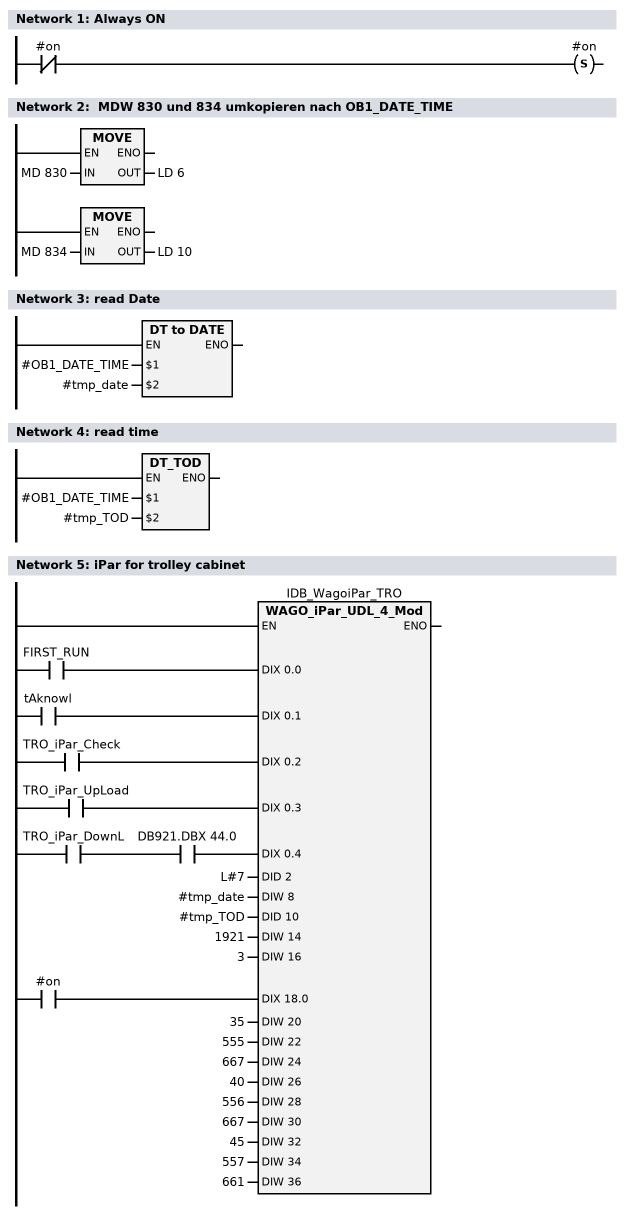
[picture p333: iPar_ServerCall networks 1-5]
NETWORK
TITLE = Always ON
      AN    #on;
      S     #on;
NETWORK
TITLE =  MDW 830 und 834 umkopieren nach OB1_DATE_TIME
      L     MD 830;
      T     LD 6;
      L     MD 834;
      T     LD 10;
NETWORK
TITLE = read Date
      CALL  "DT to DATE" (
           $1                       := #OB1_DATE_TIME,
           $2                       := #tmp_date);
      NOP   0;
NETWORK
TITLE = read time
      CALL  "DT_TOD" (
           $1                       := #OB1_DATE_TIME,
           $2                       := #tmp_TOD);
      NOP   0;
NETWORK
TITLE = iPar for trolley cabinet
      A     "FIRST_RUN";
      =     L 15.0;
      BLD   103;
      A     "tAknowl";
      =     L 15.1;
      BLD   103;
      A     "TRO_iPar_Check";
      =     L 15.2;
      BLD   103;
      A     "TRO_iPar_UpLoad";
      =     L 15.3;
      BLD   103;
      A     "TRO_iPar_DownL";
      A     DB921.DBX 44.0;
      =     L 15.4;
      BLD   103;
      A     #on;
      =     L 16.0;
      BLD   103;
      CALL  "WAGO_iPar_UDL_4_Mod" , "IDB_WagoiPar_TRO" (
           DIX 0.0                  := L 15.0,
           DIX 0.1                  := L 15.1,
           DIX 0.2                  := L 15.2,
           DIX 0.3                  := L 15.3,
           DIX 0.4                  := L 15.4,
           DID 2                    := L#7,
           DIW 8                    := #tmp_date,
           DID 10                   := #tmp_TOD,
           DIW 14                   := 1921,
           DIW 16                   := 3,
           DIX 18.0                 := L 16.0,
           DIW 20                   := 35,
           DIW 22                   := 555,
           DIW 24                   := 667,
           DIW 26                   := 40,
           DIW 28                   := 556,
           DIW 30                   := 667,
           DIW 32                   := 45,
           DIW 34                   := 557,
           DIW 36                   := 661);
      NOP   0;
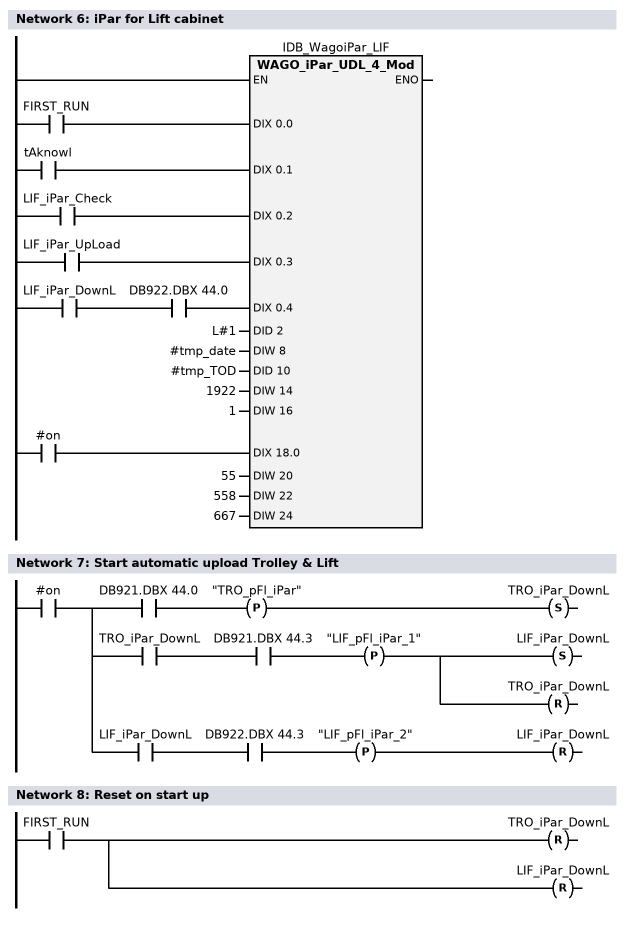
NETWORK
TITLE = iPar for Lift cabinet
      A     "FIRST_RUN";
      =     L 15.0;
      BLD   103;
      A     "tAknowl";
      =     L 15.1;
      BLD   103;
      A     "LIF_iPar_Check";
      =     L 15.2;
      BLD   103;
      A     "LIF_iPar_UpLoad";
      =     L 15.3;
      BLD   103;
      A     "LIF_iPar_DownL";
      A     DB922.DBX 44.0;
      =     L 15.4;
      BLD   103;
      A     #on;
      =     L 16.0;
      BLD   103;
      CALL  "WAGO_iPar_UDL_4_Mod" , "IDB_WagoiPar_LIF" (
           DIX 0.0                  := L 15.0,
           DIX 0.1                  := L 15.1,
           DIX 0.2                  := L 15.2,
           DIX 0.3                  := L 15.3,
           DIX 0.4                  := L 15.4,
           DID 2                    := L#1,
           DIW 8                    := #tmp_date,
           DID 10                   := #tmp_TOD,
           DIW 14                   := 1922,
           DIW 16                   := 1,
           DIX 18.0                 := L 16.0,
           DIW 20                   := 55,
           DIW 22                   := 558,
           DIW 24                   := 667);
      NOP   0;
NETWORK
TITLE = Start automatic upload Trolley & Lift
      A     #on;
      =     L 15.0;
      A     L 15.0;
      A     DB921.DBX 44.0;
      FP    "TRO_pFl_iPar";
      S     "TRO_iPar_DownL";
      A     L 15.0;
      A     "TRO_iPar_DownL";
      A     DB921.DBX 44.3;
      FP    "LIF_pFl_iPar_1";
      S     "LIF_iPar_DownL";
      R     "TRO_iPar_DownL";
      A     L 15.0;
      A     "LIF_iPar_DownL";
      A     DB922.DBX 44.3;
      FP    "LIF_pFl_iPar_2";
      R     "LIF_iPar_DownL";
NETWORK
TITLE = Reset on start up
      A     "FIRST_RUN";
      R     "TRO_iPar_DownL";
      R     "LIF_iPar_DownL";
END_FUNCTION

FUNCTION "Scan_LIF_New" : VOID	// FC 1025
TITLE = scan positions lift
VERSION : 1.0
VAR_INPUT
  in_x_ReleaseScan : BOOL ;
  in_i_LiDbNo_1 : INT ;
  in_i_LiDbNo_2 : INT ;
  in_di_NoOfDataSetsli : DINT ;
  in_di_DatSetLenghtli : DINT ;
  in_di_ActAxisPos : DINT ;
  in_di_AreaWin : DINT ;
  in_di_PosWin : DINT ;
  in_x_SelectDirection : BOOL ;	//1=right
END_VAR
VAR_OUTPUT
  out_di_Pointer : DINT ;
  out_i_DB_No : INT ;
  out_b_DB_dir_1 : BOOL ;
  out_b_DB_dir_2 : BOOL ;
  out_i_AreaNo : INT ;
  out_b_InArea : BOOL ;
  out_b_InPosHo : BOOL ;
  out_b_InPosHu : BOOL ;
  out_di_PosValHo : DINT ;
  out_di_PosValHu : DINT ;
  out_HookDataSet : UDT 102;
END_VAR
VAR_TEMP
  tmp_any_1 : ANY ;
  tmp_any_2 : ANY ;
  Save_AR1 : DWORD ;
  Save_AR2 : DWORD ;
  tmp_di_Pointer : DINT ;
  tmp_di_PosWinMinus : DINT ;
  tmp_di_PosWinPlus : DINT ;
  tmp_di_1 : DINT ;
  tmp_di_PosValHu_1 : DINT ;
  tmp_di_PosValHu_2 : DINT ;
  tmp_i_PosNo : INT ;
  tmp_i_Hooktype : INT ;
  tmp_i_DbNo : INT ;
  tmp_i_DbNo_2 : INT ;
  RetVal : INT ;
  ON : BOOL ;
  OFF : BOOL ;
  tmp_b_LoopBrake : BOOL ;
  tmp_b_1 : BOOL ;
  tmp_b_InArea_1 : BOOL ;
  tmp_b_InArea_2 : BOOL ;
  tmp_b_InPosHo_1 : BOOL ;
  tmp_b_InPosHo_2 : BOOL ;
  tmp_b_InPosHu_1 : BOOL ;
  tmp_b_InPosHu_2 : BOOL ;
  tmpHookDataSet_1 : UDT 102;
  tmpHookDataSet_2 : UDT 102;
END_VAR
BEGIN
NETWORK
TITLE = save register
      TAR1  #Save_AR1;
      TAR2  #Save_AR2;
NETWORK
TITLE = on/off
      SET;
      =     #ON;
      CLR;
      =     #OFF;
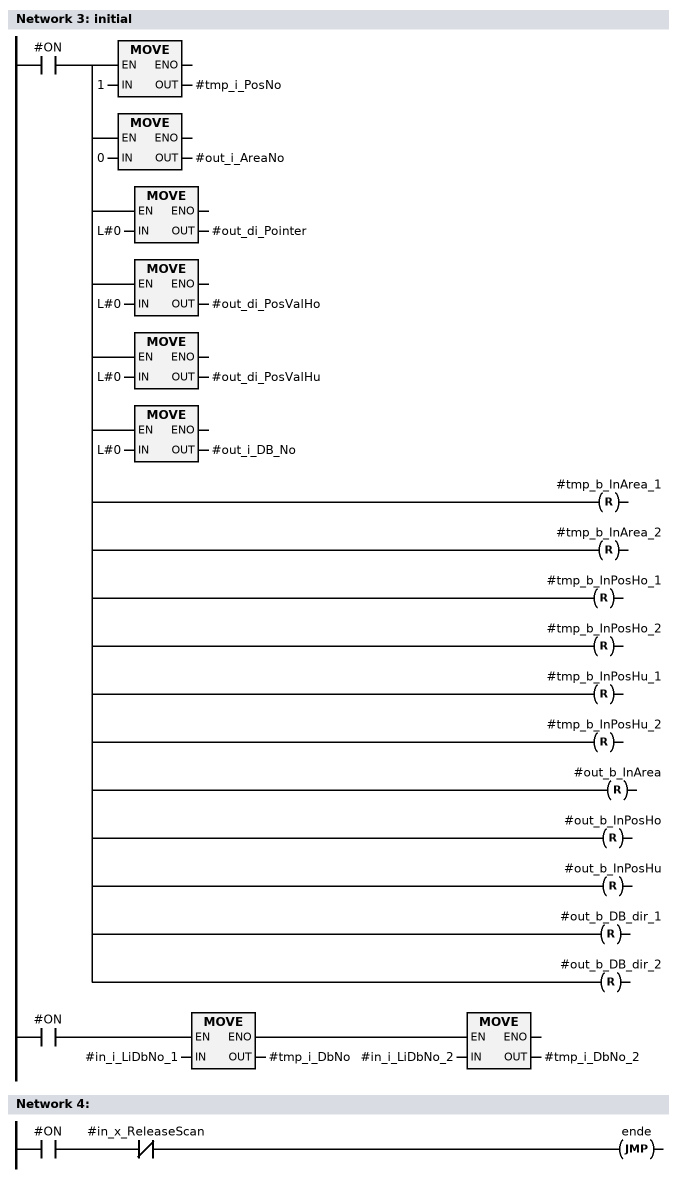
NETWORK
TITLE = initial
//#in_DbNo -> #tmp.. while "AUF DB" only with #tmp...
      A     #ON;
      =     L 176.0;
      A     L 176.0;
      JNB   _001;
      L     1;
      T     #tmp_i_PosNo;
_001: NOP   0;
      A(;
      A     L 176.0;
      JNB   _002;
      L     #in_i_LiDbNo_1;
      T     #tmp_i_DbNo;
      SET;
      SAVE;
      CLR;
_002: A     BR;
      );
      JNB   _003;
      L     #in_i_LiDbNo_2;
      T     #tmp_i_DbNo_2;
_003: NOP   0;
      A     L 176.0;
      JNB   _004;
      L     0;
      T     #out_i_AreaNo;
_004: NOP   0;
      A     L 176.0;
      JNB   _005;
      L     L#0;
      T     #out_di_Pointer;
_005: NOP   0;
      A     L 176.0;
      JNB   _006;
      L     L#0;
      T     #out_di_PosValHo;
_006: NOP   0;
      A     L 176.0;
      JNB   _007;
      L     L#0;
      T     #out_di_PosValHu;
_007: NOP   0;
      A     L 176.0;
      JNB   _008;
      L     L#0;
      T     #out_i_DB_No;
_008: NOP   0;
      A     L 176.0;
      BLD   102;
      R     #tmp_b_InArea_1;
      A     L 176.0;
      BLD   102;
      R     #tmp_b_InArea_2;
      A     L 176.0;
      BLD   102;
      R     #tmp_b_InPosHo_1;
      A     L 176.0;
      BLD   102;
      R     #tmp_b_InPosHo_2;
      A     L 176.0;
      BLD   102;
      R     #tmp_b_InPosHu_1;
      A     L 176.0;
      BLD   102;
      R     #tmp_b_InPosHu_2;
      A     L 176.0;
      BLD   102;
      R     #out_b_InArea;
      A     L 176.0;
      BLD   102;
      R     #out_b_InPosHo;
      A     L 176.0;
      BLD   102;
      R     #out_b_InPosHu;
      A     L 176.0;
      BLD   102;
      R     #out_b_DB_dir_1;
      A     L 176.0;
      BLD   102;
      R     #out_b_DB_dir_2;
NETWORK
TITLE =
      A     #ON;
      AN    #in_x_ReleaseScan;
      JC    ende;
NETWORK
TITLE = open DB
      A     #in_x_SelectDirection;
      JC    opn1;
      AN    #in_x_SelectDirection;
      JC    opn2;
      JU    ende;
opn1: OPN   DB [#tmp_i_DbNo];
      JU    opne;
opn2: OPN   DB [#tmp_i_DbNo_2];
      JU    opne;
opne: NOP   0;
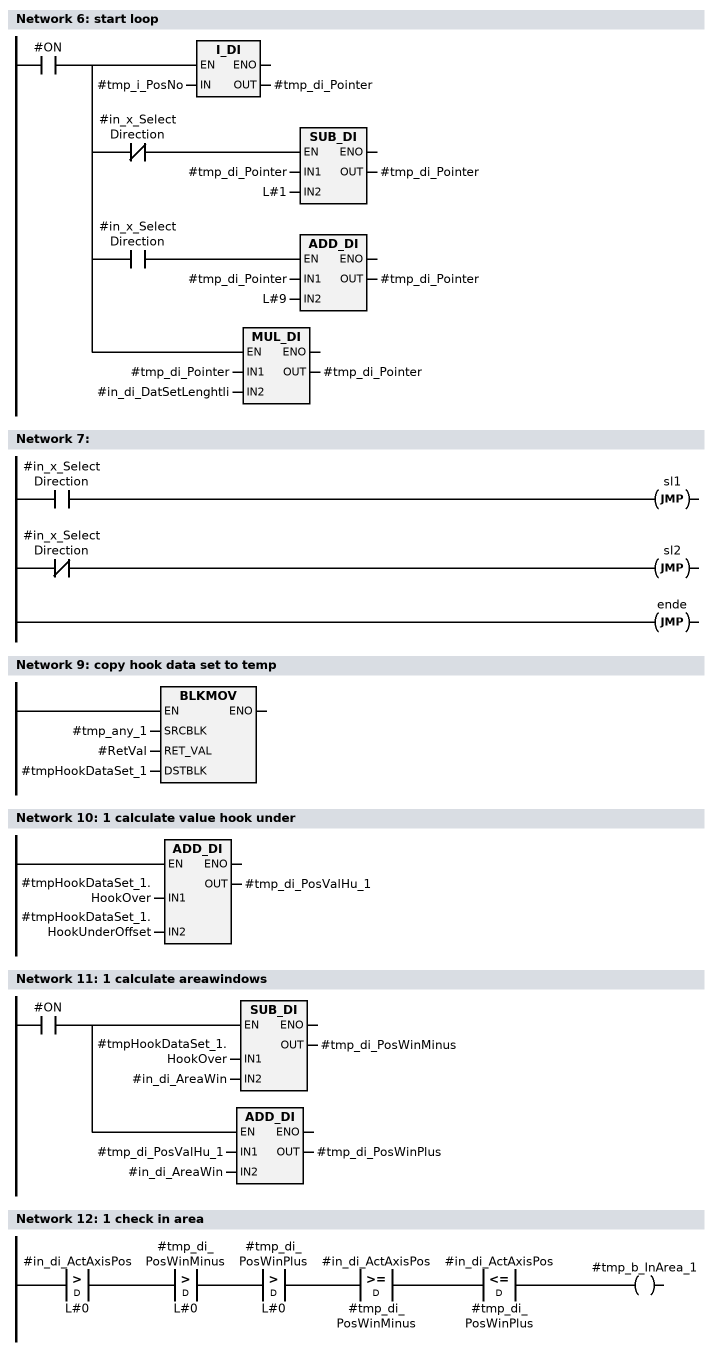
NETWORK
TITLE = start loop
//calculate Pointer to dataset
scli: A     #ON;
      =     L 176.0;
      A     L 176.0;
      JNB   _009;
      L     #tmp_i_PosNo;
      ITD;
      T     #tmp_di_Pointer;
_009: NOP   0;
      A     L 176.0;
      AN    #in_x_SelectDirection;
      JNB   _00a;
      L     #tmp_di_Pointer;
      L     L#1;
      -D;
      T     #tmp_di_Pointer;
_00a: NOP   0;
      A     L 176.0;
      A     #in_x_SelectDirection;
      JNB   _00b;
      L     #tmp_di_Pointer;
      L     L#9;
      +D;
      T     #tmp_di_Pointer;
_00b: NOP   0;
      A     L 176.0;
      JNB   _00c;
      L     #tmp_di_Pointer;
      L     #in_di_DatSetLenghtli;
      *D;
      T     #tmp_di_Pointer;
_00c: NOP   0;
NETWORK
TITLE =
      A     #in_x_SelectDirection;
      JC    sl1;
      AN    #in_x_SelectDirection;
      JC    sl2;
      NOP   0;
      JU    ende;
NETWORK
TITLE = create any-pointer to hookdataset 1
sl1:  NOP   0;
      L     W#16#1002;
      T     LW 0;
      L     56;
      T     LW 2;
      L     #tmp_i_DbNo;
      T     LW 4;
      L     #tmp_di_Pointer;
      SLD   3;
      OD    DW#16#84000000;
      T     LD 6;
NETWORK
TITLE = copy hook data set to temp
      CALL  "BLKMOV" (
           SRCBLK                   := #tmp_any_1,
           RET_VAL                  := #RetVal,
           DSTBLK                   := #tmpHookDataSet_1);
      NOP   0;
NETWORK
TITLE = 1 calculate value hook under
      L     #tmpHookDataSet_1.HookOver;
      L     #tmpHookDataSet_1.HookUnderOffset;
      +D;
      T     #tmp_di_PosValHu_1;
      NOP   0;
NETWORK
TITLE = 1 calculate areawindows
      A     #ON;
      =     L 176.0;
      A     L 176.0;
      JNB   _00d;
      L     #tmpHookDataSet_1.HookOver;
      L     #in_di_AreaWin;
      -D;
      T     #tmp_di_PosWinMinus;
_00d: NOP   0;
      A     L 176.0;
      JNB   _00e;
      L     #tmp_di_PosValHu_1;
      L     #in_di_AreaWin;
      +D;
      T     #tmp_di_PosWinPlus;
_00e: NOP   0;
NETWORK
TITLE = 1 check in area
      A(;
      L     #in_di_ActAxisPos;
      L     L#0;
      >D;
      );
      A(;
      L     #tmp_di_PosWinMinus;
      L     L#0;
      >D;
      );
      A(;
      L     #tmp_di_PosWinPlus;
      L     L#0;
      >D;
      );
      A(;
      L     #in_di_ActAxisPos;
      L     #tmp_di_PosWinMinus;
      >=D;
      );
      A(;
      L     #in_di_ActAxisPos;
      L     #tmp_di_PosWinPlus;
      <=D;
      );
      =     #tmp_b_InArea_1;
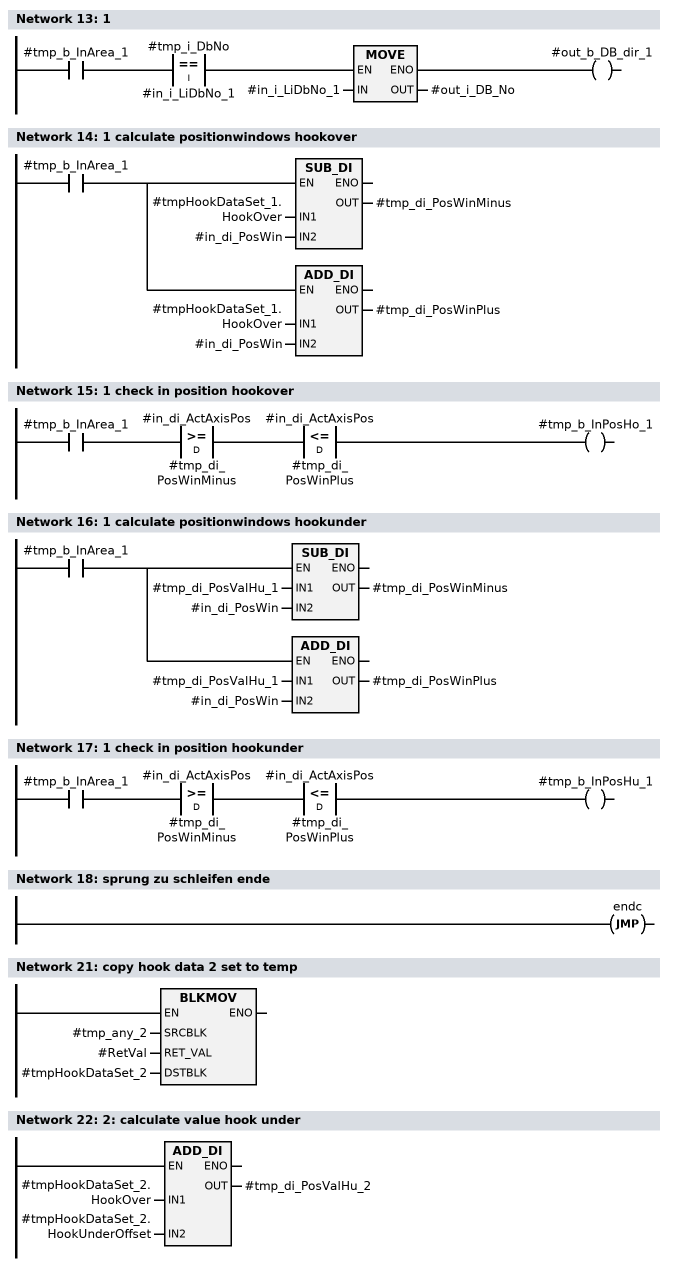
NETWORK
TITLE = 1 
      A     #tmp_b_InArea_1;
      A(;
      L     #tmp_i_DbNo;
      L     #in_i_LiDbNo_1;
      ==I;
      );
      JNB   _00f;
      L     #in_i_LiDbNo_1;
      T     #out_i_DB_No;
      SET;
      SAVE;
      CLR;
_00f: A     BR;
      =     #out_b_DB_dir_1;
NETWORK
TITLE = 1 calculate positionwindows hookover
      A     #tmp_b_InArea_1;
      =     L 176.0;
      A     L 176.0;
      JNB   _010;
      L     #tmpHookDataSet_1.HookOver;
      L     #in_di_PosWin;
      -D;
      T     #tmp_di_PosWinMinus;
_010: NOP   0;
      A     L 176.0;
      JNB   _011;
      L     #tmpHookDataSet_1.HookOver;
      L     #in_di_PosWin;
      +D;
      T     #tmp_di_PosWinPlus;
_011: NOP   0;
NETWORK
TITLE = 1 check in position hookover
      A     #tmp_b_InArea_1;
      A(;
      L     #in_di_ActAxisPos;
      L     #tmp_di_PosWinMinus;
      >=D;
      );
      A(;
      L     #in_di_ActAxisPos;
      L     #tmp_di_PosWinPlus;
      <=D;
      );
      =     #tmp_b_InPosHo_1;
NETWORK
TITLE = 1 calculate positionwindows hookunder
      A     #tmp_b_InArea_1;
      =     L 176.0;
      A     L 176.0;
      JNB   _012;
      L     #tmp_di_PosValHu_1;
      L     #in_di_PosWin;
      -D;
      T     #tmp_di_PosWinMinus;
_012: NOP   0;
      A     L 176.0;
      JNB   _013;
      L     #tmp_di_PosValHu_1;
      L     #in_di_PosWin;
      +D;
      T     #tmp_di_PosWinPlus;
_013: NOP   0;
NETWORK
TITLE = 1 check in position hookunder
      A     #tmp_b_InArea_1;
      A(;
      L     #in_di_ActAxisPos;
      L     #tmp_di_PosWinMinus;
      >=D;
      );
      A(;
      L     #in_di_ActAxisPos;
      L     #tmp_di_PosWinPlus;
      <=D;
      );
      =     #tmp_b_InPosHu_1;
NETWORK
TITLE = sprung zu schleifen ende
      JU    endc;
NETWORK
TITLE =
NETWORK
TITLE = create any-pointer to hookdataset 2
sl2:  NOP   0;
      L     W#16#1002;
      T     LW 10;
      L     56;
      T     LW 12;
      L     #tmp_i_DbNo_2;
      T     LW 14;
      L     #tmp_di_Pointer;
      SLD   3;
      OD    DW#16#84000000;
      T     LD 16;
NETWORK
TITLE = copy hook data 2 set to temp
      CALL  "BLKMOV" (
           SRCBLK                   := #tmp_any_2,
           RET_VAL                  := #RetVal,
           DSTBLK                   := #tmpHookDataSet_2);
      NOP   0;
NETWORK
TITLE = 2: calculate value hook under
      L     #tmpHookDataSet_2.HookOver;
      L     #tmpHookDataSet_2.HookUnderOffset;
      +D;
      T     #tmp_di_PosValHu_2;
      NOP   0;
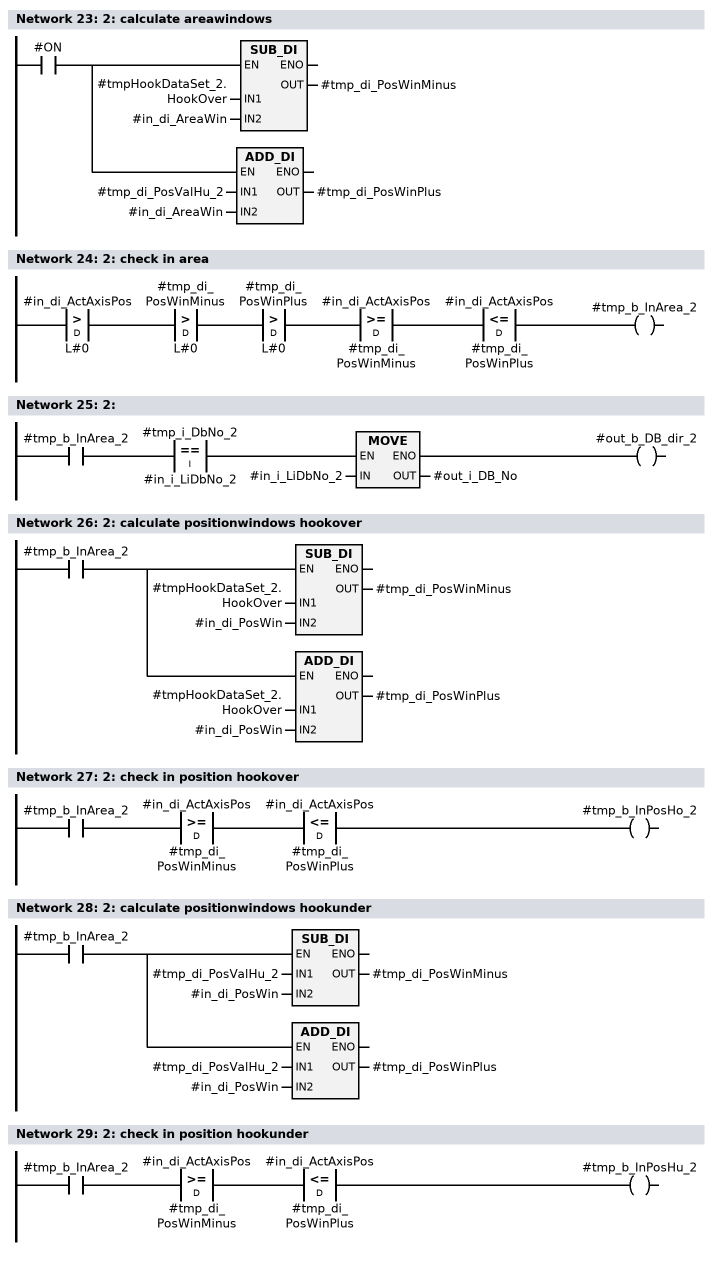
NETWORK
TITLE = 2: calculate areawindows
      A     #ON;
      =     L 176.0;
      A     L 176.0;
      JNB   _014;
      L     #tmpHookDataSet_2.HookOver;
      L     #in_di_AreaWin;
      -D;
      T     #tmp_di_PosWinMinus;
_014: NOP   0;
      A     L 176.0;
      JNB   _015;
      L     #tmp_di_PosValHu_2;
      L     #in_di_AreaWin;
      +D;
      T     #tmp_di_PosWinPlus;
_015: NOP   0;
NETWORK
TITLE = 2: check in area
      A(;
      L     #in_di_ActAxisPos;
      L     L#0;
      >D;
      );
      A(;
      L     #tmp_di_PosWinMinus;
      L     L#0;
      >D;
      );
      A(;
      L     #tmp_di_PosWinPlus;
      L     L#0;
      >D;
      );
      A(;
      L     #in_di_ActAxisPos;
      L     #tmp_di_PosWinMinus;
      >=D;
      );
      A(;
      L     #in_di_ActAxisPos;
      L     #tmp_di_PosWinPlus;
      <=D;
      );
      =     #tmp_b_InArea_2;
NETWORK
TITLE = 2:
      A     #tmp_b_InArea_2;
      A(;
      L     #tmp_i_DbNo_2;
      L     #in_i_LiDbNo_2;
      ==I;
      );
      JNB   _016;
      L     #in_i_LiDbNo_2;
      T     #out_i_DB_No;
      SET;
      SAVE;
      CLR;
_016: A     BR;
      =     #out_b_DB_dir_2;
NETWORK
TITLE = 2: calculate positionwindows hookover
      A     #tmp_b_InArea_2;
      =     L 176.0;
      A     L 176.0;
      JNB   _017;
      L     #tmpHookDataSet_2.HookOver;
      L     #in_di_PosWin;
      -D;
      T     #tmp_di_PosWinMinus;
_017: NOP   0;
      A     L 176.0;
      JNB   _018;
      L     #tmpHookDataSet_2.HookOver;
      L     #in_di_PosWin;
      +D;
      T     #tmp_di_PosWinPlus;
_018: NOP   0;
NETWORK
TITLE = 2: check in position hookover
      A     #tmp_b_InArea_2;
      A(;
      L     #in_di_ActAxisPos;
      L     #tmp_di_PosWinMinus;
      >=D;
      );
      A(;
      L     #in_di_ActAxisPos;
      L     #tmp_di_PosWinPlus;
      <=D;
      );
      =     #tmp_b_InPosHo_2;
NETWORK
TITLE = 2: calculate positionwindows hookunder
      A     #tmp_b_InArea_2;
      =     L 176.0;
      A     L 176.0;
      JNB   _019;
      L     #tmp_di_PosValHu_2;
      L     #in_di_PosWin;
      -D;
      T     #tmp_di_PosWinMinus;
_019: NOP   0;
      A     L 176.0;
      JNB   _01a;
      L     #tmp_di_PosValHu_2;
      L     #in_di_PosWin;
      +D;
      T     #tmp_di_PosWinPlus;
_01a: NOP   0;
NETWORK
TITLE = 2: check in position hookunder
      A     #tmp_b_InArea_2;
      A(;
      L     #in_di_ActAxisPos;
      L     #tmp_di_PosWinMinus;
      >=D;
      );
      A(;
      L     #in_di_ActAxisPos;
      L     #tmp_di_PosWinPlus;
      <=D;
      );
      =     #tmp_b_InPosHu_2;
NETWORK
TITLE = jump target endc
endc: NOP   0;
NETWORK
TITLE =
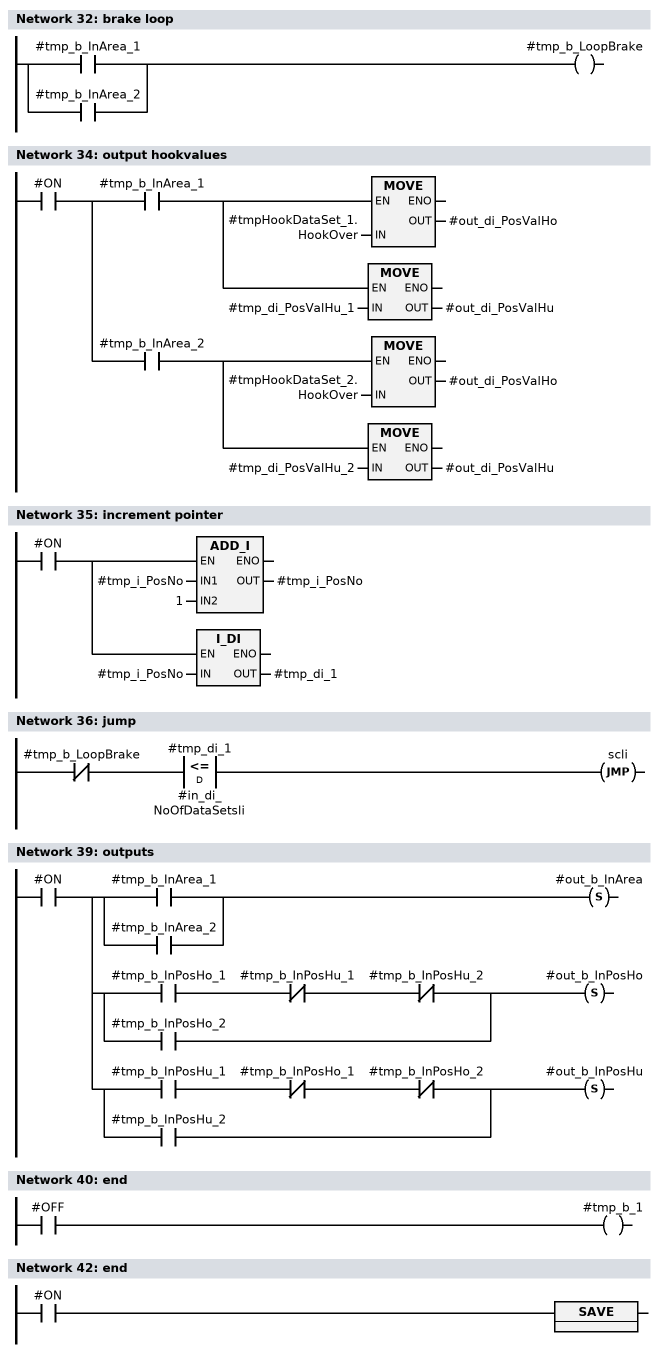
NETWORK
TITLE = brake loop
      O     #tmp_b_InArea_1;
      O     #tmp_b_InArea_2;
      =     #tmp_b_LoopBrake;
NETWORK
TITLE = output areanumber, positionnumber
//99 = Top Position
      A     #ON;
      =     L 176.0;
      A     L 176.0;
      A(;
      O     #tmp_b_InArea_1;
      O     #tmp_b_InArea_2;
      );
      =     L 176.1;
      A     L 176.1;
      JNB   _01b;
      L     #tmp_i_PosNo;
      T     #out_i_AreaNo;
_01b: NOP   0;
      A(;
      A     L 176.1;
      JNB   _01c;
      L     #tmp_i_PosNo;
      ITD;
      T     #tmp_di_1;
      SET;
      SAVE;
      CLR;
_01c: A     BR;
      );
      A(;
      L     #tmp_di_1;
      L     #in_di_NoOfDataSetsli;
      ==D;
      );
      JNB   _01d;
      L     100;
      T     #out_i_AreaNo;
_01d: NOP   0;
      A     L 176.1;
      JNB   _01e;
      L     #tmp_di_Pointer;
      T     #out_di_Pointer;
_01e: NOP   0;
      A     L 176.0;
      AN    #tmp_b_InArea_1;
      AN    #tmp_b_InArea_2;
      JNB   _01f;
      L     0;
      T     #out_i_AreaNo;
_01f: NOP   0;
NETWORK
TITLE = output hookvalues 
      A     #ON;
      =     L 176.0;
      A     L 176.0;
      A     #tmp_b_InArea_1;
      =     L 176.1;
      A     L 176.1;
      JNB   _020;
      L     #tmpHookDataSet_1.HookOver;
      T     #out_di_PosValHo;
_020: NOP   0;
      A     L 176.1;
      JNB   _021;
      L     #tmp_di_PosValHu_1;
      T     #out_di_PosValHu;
_021: NOP   0;
      A     L 176.0;
      A     #tmp_b_InArea_2;
      =     L 176.1;
      A     L 176.1;
      JNB   _022;
      L     #tmpHookDataSet_2.HookOver;
      T     #out_di_PosValHo;
_022: NOP   0;
      A     L 176.1;
      JNB   _023;
      L     #tmp_di_PosValHu_2;
      T     #out_di_PosValHu;
_023: NOP   0;
NETWORK
TITLE = increment pointer
      A     #ON;
      =     L 176.0;
      A     L 176.0;
      JNB   _024;
      L     #tmp_i_PosNo;
      L     1;
      +I;
      T     #tmp_i_PosNo;
_024: NOP   0;
      A     L 176.0;
      JNB   _025;
      L     #tmp_i_PosNo;
      ITD;
      T     #tmp_di_1;
_025: NOP   0;
NETWORK
TITLE = jump
      AN    #tmp_b_LoopBrake;
      A(;
      L     #tmp_di_1;
      L     #in_di_NoOfDataSetsli;
      <=D;
      );
      JC    scli;
NETWORK
TITLE = 1: copy hook data to out
      A     #tmp_b_InArea_1;
      =     L 176.0;
      A(;
      A     L 176.0;
      JNB   _026;
      L     #tmpHookDataSet_1.HookOver;
      BLD   5;
      T     LD 179;
      TAK;
      T     LD 183;
      L     P##out_HookDataSet;
      LAR1;
      L     W [AR1,P#0.0];
      T     LW 177;
      OPN   DB [LW 177];
      L     D [AR1,P#2.0];
      LAR1;
      L     LD 183;
      L     LD 179;
      T     D [AR1,P#0.0];
      SET;
      SAVE;
      CLR;
_026: A     BR;
      );
      JNB   _027;
      L     #tmpHookDataSet_1.HookUnderOffset;
      BLD   5;
      T     LD 179;
      TAK;
      T     LD 183;
      L     P##out_HookDataSet;
      LAR1;
      L     W [AR1,P#0.0];
      T     LW 177;
      OPN   DB [LW 177];
      L     D [AR1,P#2.0];
      LAR1;
      L     LD 183;
      L     LD 179;
      T     D [AR1,P#4.0];
_027: NOP   0;
      A(;
      A(;
      A     L 176.0;
      JNB   _028;
      L     #tmpHookDataSet_1.TelPos_1.TelPos;
      BLD   5;
      T     LD 179;
      TAK;
      T     LD 183;
      L     P##out_HookDataSet;
      LAR1;
      L     W [AR1,P#0.0];
      T     LW 177;
      OPN   DB [LW 177];
      L     D [AR1,P#2.0];
      LAR1;
      L     LD 183;
      L     LD 179;
      T     D [AR1,P#18.0];
      SET;
      SAVE;
      CLR;
_028: A     BR;
      );
      JNB   _029;
      L     #tmpHookDataSet_1.TelPos_2.TelPos;
      BLD   5;
      T     LD 179;
      TAK;
      T     LD 183;
      L     P##out_HookDataSet;
      LAR1;
      L     W [AR1,P#0.0];
      T     LW 177;
      OPN   DB [LW 177];
      L     D [AR1,P#2.0];
      LAR1;
      L     LD 183;
      L     LD 179;
      T     D [AR1,P#34.0];
      SET;
      SAVE;
      CLR;
_029: A     BR;
      );
      JNB   _02a;
      L     #tmpHookDataSet_1.TelPos_3.TelPos;
      BLD   5;
      T     LD 179;
      TAK;
      T     LD 183;
      L     P##out_HookDataSet;
      LAR1;
      L     W [AR1,P#0.0];
      T     LW 177;
      OPN   DB [LW 177];
      L     D [AR1,P#2.0];
      LAR1;
      L     LD 183;
      L     LD 179;
      T     D [AR1,P#50.0];
_02a: NOP   0;
      A(;
      A(;
      A     L 176.0;
      JNB   _02b;
      L     #tmpHookDataSet_1.TelPos_1.TotLengthMin;
      BLD   5;
      T     LD 179;
      TAK;
      T     LD 183;
      L     P##out_HookDataSet;
      LAR1;
      L     W [AR1,P#0.0];
      T     LW 177;
      OPN   DB [LW 177];
      L     D [AR1,P#2.0];
      LAR1;
      L     LD 183;
      L     LD 179;
      T     W [AR1,P#10.0];
      SET;
      SAVE;
      CLR;
_02b: A     BR;
      );
      JNB   _02c;
      L     #tmpHookDataSet_1.TelPos_1.TotLengthMax;
      BLD   5;
      T     LD 179;
      TAK;
      T     LD 183;
      L     P##out_HookDataSet;
      LAR1;
      L     W [AR1,P#0.0];
      T     LW 177;
      OPN   DB [LW 177];
      L     D [AR1,P#2.0];
      LAR1;
      L     LD 183;
      L     LD 179;
      T     W [AR1,P#12.0];
      SET;
      SAVE;
      CLR;
_02c: A     BR;
      );
      JNB   _02d;
      L     #tmpHookDataSet_1.TelPos_1.FaceLengthMax;
      BLD   5;
      T     LD 179;
      TAK;
      T     LD 183;
      L     P##out_HookDataSet;
      LAR1;
      L     W [AR1,P#0.0];
      T     LW 177;
      OPN   DB [LW 177];
      L     D [AR1,P#2.0];
      LAR1;
      L     LD 183;
      L     LD 179;
      T     W [AR1,P#14.0];
_02d: NOP   0;
      A(;
      A(;
      A     L 176.0;
      JNB   _02e;
      L     #tmpHookDataSet_1.TelPos_1.CircumMax;
      BLD   5;
      T     LD 179;
      TAK;
      T     LD 183;
      L     P##out_HookDataSet;
      LAR1;
      L     W [AR1,P#0.0];
      T     LW 177;
      OPN   DB [LW 177];
      L     D [AR1,P#2.0];
      LAR1;
      L     LD 183;
      L     LD 179;
      T     W [AR1,P#16.0];
      SET;
      SAVE;
      CLR;
_02e: A     BR;
      );
      JNB   _02f;
      L     #tmpHookDataSet_1.TelPos_1.HookType;
      BLD   5;
      T     LD 179;
      TAK;
      T     LD 183;
      L     P##out_HookDataSet;
      LAR1;
      L     W [AR1,P#0.0];
      T     LW 177;
      OPN   DB [LW 177];
      L     D [AR1,P#2.0];
      LAR1;
      L     LD 183;
      L     LD 179;
      T     W [AR1,P#8.0];
      SET;
      SAVE;
      CLR;
_02f: A     BR;
      );
      JNB   _030;
      L     #tmpHookDataSet_1.TelPos_1.Reserve1;
      BLD   5;
      T     LD 179;
      TAK;
      T     LD 183;
      L     P##out_HookDataSet;
      LAR1;
      L     W [AR1,P#0.0];
      T     LW 177;
      OPN   DB [LW 177];
      L     D [AR1,P#2.0];
      LAR1;
      L     LD 183;
      L     LD 179;
      T     W [AR1,P#22.0];
_030: NOP   0;
      A(;
      A(;
      A     L 176.0;
      JNB   _031;
      L     #tmpHookDataSet_1.TelPos_2.TotLengthMin;
      BLD   5;
      T     LD 179;
      TAK;
      T     LD 183;
      L     P##out_HookDataSet;
      LAR1;
      L     W [AR1,P#0.0];
      T     LW 177;
      OPN   DB [LW 177];
      L     D [AR1,P#2.0];
      LAR1;
      L     LD 183;
      L     LD 179;
      T     W [AR1,P#26.0];
      SET;
      SAVE;
      CLR;
_031: A     BR;
      );
      JNB   _032;
      L     #tmpHookDataSet_1.TelPos_2.TotLengthMax;
      BLD   5;
      T     LD 179;
      TAK;
      T     LD 183;
      L     P##out_HookDataSet;
      LAR1;
      L     W [AR1,P#0.0];
      T     LW 177;
      OPN   DB [LW 177];
      L     D [AR1,P#2.0];
      LAR1;
      L     LD 183;
      L     LD 179;
      T     W [AR1,P#28.0];
      SET;
      SAVE;
      CLR;
_032: A     BR;
      );
      JNB   _033;
      L     #tmpHookDataSet_1.TelPos_2.FaceLengthMax;
      BLD   5;
      T     LD 179;
      TAK;
      T     LD 183;
      L     P##out_HookDataSet;
      LAR1;
      L     W [AR1,P#0.0];
      T     LW 177;
      OPN   DB [LW 177];
      L     D [AR1,P#2.0];
      LAR1;
      L     LD 183;
      L     LD 179;
      T     W [AR1,P#30.0];
_033: NOP   0;
      A(;
      A(;
      A     L 176.0;
      JNB   _034;
      L     #tmpHookDataSet_1.TelPos_2.CircumMax;
      BLD   5;
      T     LD 179;
      TAK;
      T     LD 183;
      L     P##out_HookDataSet;
      LAR1;
      L     W [AR1,P#0.0];
      T     LW 177;
      OPN   DB [LW 177];
      L     D [AR1,P#2.0];
      LAR1;
      L     LD 183;
      L     LD 179;
      T     W [AR1,P#32.0];
      SET;
      SAVE;
      CLR;
_034: A     BR;
      );
      JNB   _035;
      L     #tmpHookDataSet_1.TelPos_2.HookType;
      BLD   5;
      T     LD 179;
      TAK;
      T     LD 183;
      L     P##out_HookDataSet;
      LAR1;
      L     W [AR1,P#0.0];
      T     LW 177;
      OPN   DB [LW 177];
      L     D [AR1,P#2.0];
      LAR1;
      L     LD 183;
      L     LD 179;
      T     W [AR1,P#24.0];
      SET;
      SAVE;
      CLR;
_035: A     BR;
      );
      JNB   _036;
      L     #tmpHookDataSet_1.TelPos_2.Reserve1;
      BLD   5;
      T     LD 179;
      TAK;
      T     LD 183;
      L     P##out_HookDataSet;
      LAR1;
      L     W [AR1,P#0.0];
      T     LW 177;
      OPN   DB [LW 177];
      L     D [AR1,P#2.0];
      LAR1;
      L     LD 183;
      L     LD 179;
      T     W [AR1,P#38.0];
_036: NOP   0;
      A(;
      A(;
      A     L 176.0;
      JNB   _037;
      L     #tmpHookDataSet_1.TelPos_3.TotLengthMin;
      BLD   5;
      T     LD 179;
      TAK;
      T     LD 183;
      L     P##out_HookDataSet;
      LAR1;
      L     W [AR1,P#0.0];
      T     LW 177;
      OPN   DB [LW 177];
      L     D [AR1,P#2.0];
      LAR1;
      L     LD 183;
      L     LD 179;
      T     W [AR1,P#42.0];
      SET;
      SAVE;
      CLR;
_037: A     BR;
      );
      JNB   _038;
      L     #tmpHookDataSet_1.TelPos_3.TotLengthMax;
      BLD   5;
      T     LD 179;
      TAK;
      T     LD 183;
      L     P##out_HookDataSet;
      LAR1;
      L     W [AR1,P#0.0];
      T     LW 177;
      OPN   DB [LW 177];
      L     D [AR1,P#2.0];
      LAR1;
      L     LD 183;
      L     LD 179;
      T     W [AR1,P#44.0];
      SET;
      SAVE;
      CLR;
_038: A     BR;
      );
      JNB   _039;
      L     #tmpHookDataSet_1.TelPos_3.FaceLengthMax;
      BLD   5;
      T     LD 179;
      TAK;
      T     LD 183;
      L     P##out_HookDataSet;
      LAR1;
      L     W [AR1,P#0.0];
      T     LW 177;
      OPN   DB [LW 177];
      L     D [AR1,P#2.0];
      LAR1;
      L     LD 183;
      L     LD 179;
      T     W [AR1,P#46.0];
_039: NOP   0;
      A(;
      A(;
      A     L 176.0;
      JNB   _03a;
      L     #tmpHookDataSet_1.TelPos_3.CircumMax;
      BLD   5;
      T     LD 179;
      TAK;
      T     LD 183;
      L     P##out_HookDataSet;
      LAR1;
      L     W [AR1,P#0.0];
      T     LW 177;
      OPN   DB [LW 177];
      L     D [AR1,P#2.0];
      LAR1;
      L     LD 183;
      L     LD 179;
      T     W [AR1,P#48.0];
      SET;
      SAVE;
      CLR;
_03a: A     BR;
      );
      JNB   _03b;
      L     #tmpHookDataSet_1.TelPos_3.HookType;
      BLD   5;
      T     LD 179;
      TAK;
      T     LD 183;
      L     P##out_HookDataSet;
      LAR1;
      L     W [AR1,P#0.0];
      T     LW 177;
      OPN   DB [LW 177];
      L     D [AR1,P#2.0];
      LAR1;
      L     LD 183;
      L     LD 179;
      T     W [AR1,P#40.0];
      SET;
      SAVE;
      CLR;
_03b: A     BR;
      );
      JNB   _03c;
      L     #tmpHookDataSet_1.TelPos_3.Reserve1;
      BLD   5;
      T     LD 179;
      TAK;
      T     LD 183;
      L     P##out_HookDataSet;
      LAR1;
      L     W [AR1,P#0.0];
      T     LW 177;
      OPN   DB [LW 177];
      L     D [AR1,P#2.0];
      LAR1;
      L     LD 183;
      L     LD 179;
      T     W [AR1,P#54.0];
_03c: NOP   0;
NETWORK
TITLE = 2: copy hook data to out
      A     #tmp_b_InArea_2;
      =     L 176.0;
      A(;
      A     L 176.0;
      JNB   _03d;
      L     #tmpHookDataSet_2.HookOver;
      BLD   5;
      T     LD 179;
      TAK;
      T     LD 183;
      L     P##out_HookDataSet;
      LAR1;
      L     W [AR1,P#0.0];
      T     LW 177;
      OPN   DB [LW 177];
      L     D [AR1,P#2.0];
      LAR1;
      L     LD 183;
      L     LD 179;
      T     D [AR1,P#0.0];
      SET;
      SAVE;
      CLR;
_03d: A     BR;
      );
      JNB   _03e;
      L     #tmpHookDataSet_2.HookUnderOffset;
      BLD   5;
      T     LD 179;
      TAK;
      T     LD 183;
      L     P##out_HookDataSet;
      LAR1;
      L     W [AR1,P#0.0];
      T     LW 177;
      OPN   DB [LW 177];
      L     D [AR1,P#2.0];
      LAR1;
      L     LD 183;
      L     LD 179;
      T     D [AR1,P#4.0];
_03e: NOP   0;
      A(;
      A(;
      A     L 176.0;
      JNB   _03f;
      L     #tmpHookDataSet_2.TelPos_1.TelPos;
      BLD   5;
      T     LD 179;
      TAK;
      T     LD 183;
      L     P##out_HookDataSet;
      LAR1;
      L     W [AR1,P#0.0];
      T     LW 177;
      OPN   DB [LW 177];
      L     D [AR1,P#2.0];
      LAR1;
      L     LD 183;
      L     LD 179;
      T     D [AR1,P#18.0];
      SET;
      SAVE;
      CLR;
_03f: A     BR;
      );
      JNB   _040;
      L     #tmpHookDataSet_2.TelPos_2.TelPos;
      BLD   5;
      T     LD 179;
      TAK;
      T     LD 183;
      L     P##out_HookDataSet;
      LAR1;
      L     W [AR1,P#0.0];
      T     LW 177;
      OPN   DB [LW 177];
      L     D [AR1,P#2.0];
      LAR1;
      L     LD 183;
      L     LD 179;
      T     D [AR1,P#34.0];
      SET;
      SAVE;
      CLR;
_040: A     BR;
      );
      JNB   _041;
      L     #tmpHookDataSet_2.TelPos_3.TelPos;
      BLD   5;
      T     LD 179;
      TAK;
      T     LD 183;
      L     P##out_HookDataSet;
      LAR1;
      L     W [AR1,P#0.0];
      T     LW 177;
      OPN   DB [LW 177];
      L     D [AR1,P#2.0];
      LAR1;
      L     LD 183;
      L     LD 179;
      T     D [AR1,P#50.0];
_041: NOP   0;
      A(;
      A(;
      A     L 176.0;
      JNB   _042;
      L     #tmpHookDataSet_2.TelPos_1.TotLengthMin;
      BLD   5;
      T     LD 179;
      TAK;
      T     LD 183;
      L     P##out_HookDataSet;
      LAR1;
      L     W [AR1,P#0.0];
      T     LW 177;
      OPN   DB [LW 177];
      L     D [AR1,P#2.0];
      LAR1;
      L     LD 183;
      L     LD 179;
      T     W [AR1,P#10.0];
      SET;
      SAVE;
      CLR;
_042: A     BR;
      );
      JNB   _043;
      L     #tmpHookDataSet_2.TelPos_1.TotLengthMax;
      BLD   5;
      T     LD 179;
      TAK;
      T     LD 183;
      L     P##out_HookDataSet;
      LAR1;
      L     W [AR1,P#0.0];
      T     LW 177;
      OPN   DB [LW 177];
      L     D [AR1,P#2.0];
      LAR1;
      L     LD 183;
      L     LD 179;
      T     W [AR1,P#12.0];
      SET;
      SAVE;
      CLR;
_043: A     BR;
      );
      JNB   _044;
      L     #tmpHookDataSet_2.TelPos_1.FaceLengthMax;
      BLD   5;
      T     LD 179;
      TAK;
      T     LD 183;
      L     P##out_HookDataSet;
      LAR1;
      L     W [AR1,P#0.0];
      T     LW 177;
      OPN   DB [LW 177];
      L     D [AR1,P#2.0];
      LAR1;
      L     LD 183;
      L     LD 179;
      T     W [AR1,P#14.0];
_044: NOP   0;
      A(;
      A(;
      A     L 176.0;
      JNB   _045;
      L     #tmpHookDataSet_2.TelPos_1.CircumMax;
      BLD   5;
      T     LD 179;
      TAK;
      T     LD 183;
      L     P##out_HookDataSet;
      LAR1;
      L     W [AR1,P#0.0];
      T     LW 177;
      OPN   DB [LW 177];
      L     D [AR1,P#2.0];
      LAR1;
      L     LD 183;
      L     LD 179;
      T     W [AR1,P#16.0];
      SET;
      SAVE;
      CLR;
_045: A     BR;
      );
      JNB   _046;
      L     #tmpHookDataSet_2.TelPos_1.HookType;
      BLD   5;
      T     LD 179;
      TAK;
      T     LD 183;
      L     P##out_HookDataSet;
      LAR1;
      L     W [AR1,P#0.0];
      T     LW 177;
      OPN   DB [LW 177];
      L     D [AR1,P#2.0];
      LAR1;
      L     LD 183;
      L     LD 179;
      T     W [AR1,P#8.0];
      SET;
      SAVE;
      CLR;
_046: A     BR;
      );
      JNB   _047;
      L     #tmpHookDataSet_2.TelPos_1.Reserve1;
      BLD   5;
      T     LD 179;
      TAK;
      T     LD 183;
      L     P##out_HookDataSet;
      LAR1;
      L     W [AR1,P#0.0];
      T     LW 177;
      OPN   DB [LW 177];
      L     D [AR1,P#2.0];
      LAR1;
      L     LD 183;
      L     LD 179;
      T     W [AR1,P#22.0];
_047: NOP   0;
      A(;
      A(;
      A     L 176.0;
      JNB   _048;
      L     #tmpHookDataSet_2.TelPos_2.TotLengthMin;
      BLD   5;
      T     LD 179;
      TAK;
      T     LD 183;
      L     P##out_HookDataSet;
      LAR1;
      L     W [AR1,P#0.0];
      T     LW 177;
      OPN   DB [LW 177];
      L     D [AR1,P#2.0];
      LAR1;
      L     LD 183;
      L     LD 179;
      T     W [AR1,P#26.0];
      SET;
      SAVE;
      CLR;
_048: A     BR;
      );
      JNB   _049;
      L     #tmpHookDataSet_2.TelPos_2.TotLengthMax;
      BLD   5;
      T     LD 179;
      TAK;
      T     LD 183;
      L     P##out_HookDataSet;
      LAR1;
      L     W [AR1,P#0.0];
      T     LW 177;
      OPN   DB [LW 177];
      L     D [AR1,P#2.0];
      LAR1;
      L     LD 183;
      L     LD 179;
      T     W [AR1,P#28.0];
      SET;
      SAVE;
      CLR;
_049: A     BR;
      );
      JNB   _04a;
      L     #tmpHookDataSet_2.TelPos_2.FaceLengthMax;
      BLD   5;
      T     LD 179;
      TAK;
      T     LD 183;
      L     P##out_HookDataSet;
      LAR1;
      L     W [AR1,P#0.0];
      T     LW 177;
      OPN   DB [LW 177];
      L     D [AR1,P#2.0];
      LAR1;
      L     LD 183;
      L     LD 179;
      T     W [AR1,P#30.0];
_04a: NOP   0;
      A(;
      A(;
      A     L 176.0;
      JNB   _04b;
      L     #tmpHookDataSet_2.TelPos_2.CircumMax;
      BLD   5;
      T     LD 179;
      TAK;
      T     LD 183;
      L     P##out_HookDataSet;
      LAR1;
      L     W [AR1,P#0.0];
      T     LW 177;
      OPN   DB [LW 177];
      L     D [AR1,P#2.0];
      LAR1;
      L     LD 183;
      L     LD 179;
      T     W [AR1,P#32.0];
      SET;
      SAVE;
      CLR;
_04b: A     BR;
      );
      JNB   _04c;
      L     #tmpHookDataSet_2.TelPos_2.HookType;
      BLD   5;
      T     LD 179;
      TAK;
      T     LD 183;
      L     P##out_HookDataSet;
      LAR1;
      L     W [AR1,P#0.0];
      T     LW 177;
      OPN   DB [LW 177];
      L     D [AR1,P#2.0];
      LAR1;
      L     LD 183;
      L     LD 179;
      T     W [AR1,P#24.0];
      SET;
      SAVE;
      CLR;
_04c: A     BR;
      );
      JNB   _04d;
      L     #tmpHookDataSet_2.TelPos_2.Reserve1;
      BLD   5;
      T     LD 179;
      TAK;
      T     LD 183;
      L     P##out_HookDataSet;
      LAR1;
      L     W [AR1,P#0.0];
      T     LW 177;
      OPN   DB [LW 177];
      L     D [AR1,P#2.0];
      LAR1;
      L     LD 183;
      L     LD 179;
      T     W [AR1,P#38.0];
_04d: NOP   0;
      A(;
      A(;
      A     L 176.0;
      JNB   _04e;
      L     #tmpHookDataSet_2.TelPos_3.TotLengthMin;
      BLD   5;
      T     LD 179;
      TAK;
      T     LD 183;
      L     P##out_HookDataSet;
      LAR1;
      L     W [AR1,P#0.0];
      T     LW 177;
      OPN   DB [LW 177];
      L     D [AR1,P#2.0];
      LAR1;
      L     LD 183;
      L     LD 179;
      T     W [AR1,P#42.0];
      SET;
      SAVE;
      CLR;
_04e: A     BR;
      );
      JNB   _04f;
      L     #tmpHookDataSet_2.TelPos_3.TotLengthMax;
      BLD   5;
      T     LD 179;
      TAK;
      T     LD 183;
      L     P##out_HookDataSet;
      LAR1;
      L     W [AR1,P#0.0];
      T     LW 177;
      OPN   DB [LW 177];
      L     D [AR1,P#2.0];
      LAR1;
      L     LD 183;
      L     LD 179;
      T     W [AR1,P#44.0];
      SET;
      SAVE;
      CLR;
_04f: A     BR;
      );
      JNB   _050;
      L     #tmpHookDataSet_2.TelPos_3.FaceLengthMax;
      BLD   5;
      T     LD 179;
      TAK;
      T     LD 183;
      L     P##out_HookDataSet;
      LAR1;
      L     W [AR1,P#0.0];
      T     LW 177;
      OPN   DB [LW 177];
      L     D [AR1,P#2.0];
      LAR1;
      L     LD 183;
      L     LD 179;
      T     W [AR1,P#46.0];
_050: NOP   0;
      A(;
      A(;
      A     L 176.0;
      JNB   _051;
      L     #tmpHookDataSet_2.TelPos_3.CircumMax;
      BLD   5;
      T     LD 179;
      TAK;
      T     LD 183;
      L     P##out_HookDataSet;
      LAR1;
      L     W [AR1,P#0.0];
      T     LW 177;
      OPN   DB [LW 177];
      L     D [AR1,P#2.0];
      LAR1;
      L     LD 183;
      L     LD 179;
      T     W [AR1,P#48.0];
      SET;
      SAVE;
      CLR;
_051: A     BR;
      );
      JNB   _052;
      L     #tmpHookDataSet_2.TelPos_3.HookType;
      BLD   5;
      T     LD 179;
      TAK;
      T     LD 183;
      L     P##out_HookDataSet;
      LAR1;
      L     W [AR1,P#0.0];
      T     LW 177;
      OPN   DB [LW 177];
      L     D [AR1,P#2.0];
      LAR1;
      L     LD 183;
      L     LD 179;
      T     W [AR1,P#40.0];
      SET;
      SAVE;
      CLR;
_052: A     BR;
      );
      JNB   _053;
      L     #tmpHookDataSet_2.TelPos_3.Reserve1;
      BLD   5;
      T     LD 179;
      TAK;
      T     LD 183;
      L     P##out_HookDataSet;
      LAR1;
      L     W [AR1,P#0.0];
      T     LW 177;
      OPN   DB [LW 177];
      L     D [AR1,P#2.0];
      LAR1;
      L     LD 183;
      L     LD 179;
      T     W [AR1,P#54.0];
_053: NOP   0;
NETWORK
TITLE = outputs
      A     #ON;
      =     L 176.0;
      A     L 176.0;
      A(;
      O     #tmp_b_InArea_1;
      O     #tmp_b_InArea_2;
      );
      S     #out_b_InArea;
      A     L 176.0;
      A(;
      A     #tmp_b_InPosHo_1;
      AN    #tmp_b_InPosHu_1;
      AN    #tmp_b_InPosHu_2;
      O     #tmp_b_InPosHo_2;
      );
      S     #out_b_InPosHo;
      A     L 176.0;
      A(;
      A     #tmp_b_InPosHu_1;
      AN    #tmp_b_InPosHo_1;
      AN    #tmp_b_InPosHo_2;
      O     #tmp_b_InPosHu_2;
      );
      S     #out_b_InPosHu;
NETWORK
TITLE = end
ende: A     #OFF;
      =     #tmp_b_1;
NETWORK
TITLE = restore register
      LAR1  #Save_AR1;
      LAR2  #Save_AR2;
NETWORK
TITLE = end
      A     #ON;
      SAVE;
END_FUNCTION

FUNCTION "Scan_LIF_Man_New" : VOID	// FC 1026
TITLE = scan positions LIFt manual mode
VERSION : 1.0
VAR_INPUT
  in_b_release : BOOL ;
  in_i_DBNo : INT ;
  in_i_NoOfDataSets : INT ;
  in_i_DatSetLenght : INT ;
  in_i_DataStartByte : INT ;
  in_di_ActAxisPos : DINT ;
  in_b_Occupied : BOOL ;
  in_di_PosValMin : DINT ;
  in_di_PosValMax : DINT ;
  in_b_SelectDirection : BOOL ;	//1=right
END_VAR
VAR_OUTPUT
  out_di_PrevPos : DINT ;
  out_di_NextPos : DINT ;
  out_di_MinPos : DINT ;
  out_di_MaxPos : DINT ;
END_VAR
VAR_TEMP
  Save_AR1 : DWORD ;
  Save_AR2 : DWORD ;
  tmp_di_1 : DINT ;
  tmp_di_Pointer : DINT ;
  tmp_di_ChkPosValHo_1 : DINT ;
  tmp_di_ChkPosValHo_2 : DINT ;
  tmp_di_ChkPosValHu_1 : DINT ;
  tmp_di_ChkPosValHu_2 : DINT ;
  tmp_di_ChkPosVal_1 : DINT ;
  tmp_di_ChkPosVal_2 : DINT ;
  tmp_di_PosData : DINT ;
  tmp_di_PosDataPlus : DINT ;
  tmp_di_PosDataMinus : DINT ;
  tmp_di_PosDataLow : DINT ;
  tmp_di_PosDataHigh : DINT ;
  tmp_di_PrevPos : DINT ;
  tmp_di_NextPos : DINT ;
  tmp_i_Counter : INT ;
  tmp_i_DBNo : INT ;
  tmp_i_NoOfDataSets : INT ;
  tmp_i : INT ;
  ON : BOOL ;
  OFF : BOOL ;
  tmp_b_1 : BOOL ;
  dataSets : INT ;
END_VAR
BEGIN
NETWORK
TITLE = save register
      TAR1  #Save_AR1;
      TAR2  #Save_AR2;
NETWORK
TITLE = on/off
      SET;
      =     #ON;
      CLR;
      =     #OFF;
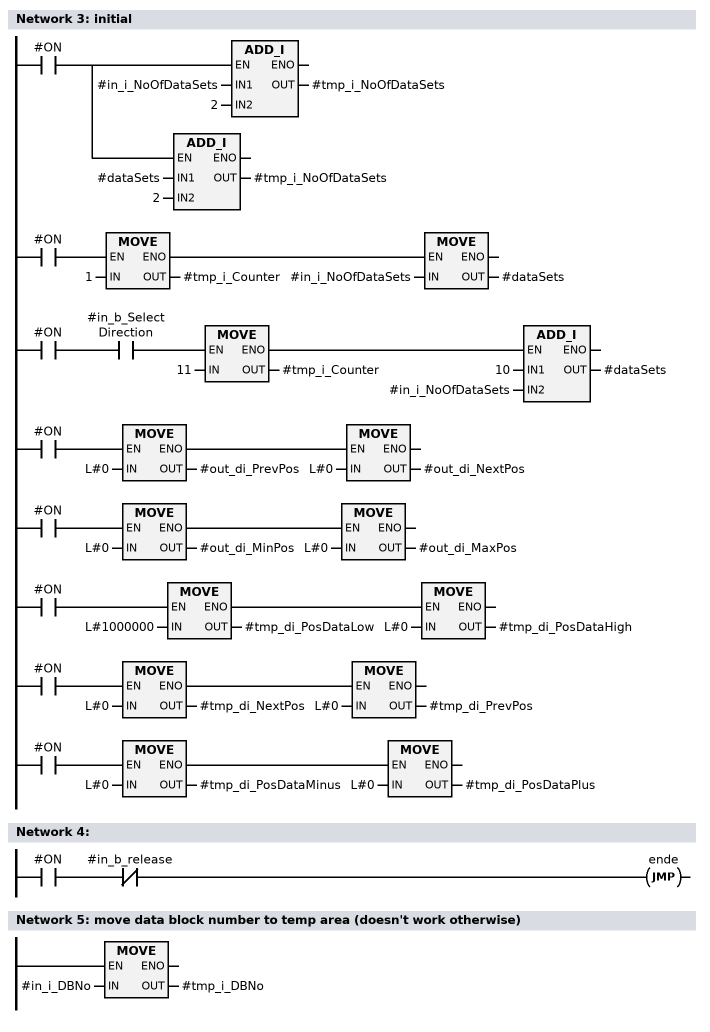
NETWORK
TITLE = initial
//set loopcounter to 0
//reset outputs
      A     #ON;
      =     L 80.0;
      A(;
      A     L 80.0;
      JNB   _001;
      L     1;
      T     #tmp_i_Counter;
      SET;
      SAVE;
      CLR;
_001: A     BR;
      );
      JNB   _002;
      L     #in_i_NoOfDataSets;
      T     #dataSets;
_002: NOP   0;
      A(;
      A     L 80.0;
      A     #in_b_SelectDirection;
      JNB   _003;
      L     11;
      T     #tmp_i_Counter;
      SET;
      SAVE;
      CLR;
_003: A     BR;
      );
      JNB   _004;
      L     10;
      L     #in_i_NoOfDataSets;
      +I;
      T     #dataSets;
_004: NOP   0;
      A(;
      A     L 80.0;
      JNB   _005;
      L     L#0;
      T     #out_di_PrevPos;
      SET;
      SAVE;
      CLR;
_005: A     BR;
      );
      JNB   _006;
      L     L#0;
      T     #out_di_NextPos;
_006: NOP   0;
      A(;
      A     L 80.0;
      JNB   _007;
      L     L#0;
      T     #out_di_MinPos;
      SET;
      SAVE;
      CLR;
_007: A     BR;
      );
      JNB   _008;
      L     L#0;
      T     #out_di_MaxPos;
_008: NOP   0;
      A(;
      A     L 80.0;
      JNB   _009;
      L     L#1000000;
      T     #tmp_di_PosDataLow;
      SET;
      SAVE;
      CLR;
_009: A     BR;
      );
      JNB   _00a;
      L     L#0;
      T     #tmp_di_PosDataHigh;
_00a: NOP   0;
      A(;
      A     L 80.0;
      JNB   _00b;
      L     L#0;
      T     #tmp_di_NextPos;
      SET;
      SAVE;
      CLR;
_00b: A     BR;
      );
      JNB   _00c;
      L     L#0;
      T     #tmp_di_PrevPos;
_00c: NOP   0;
      A(;
      A     L 80.0;
      JNB   _00d;
      L     L#0;
      T     #tmp_di_PosDataMinus;
      SET;
      SAVE;
      CLR;
_00d: A     BR;
      );
      JNB   _00e;
      L     L#0;
      T     #tmp_di_PosDataPlus;
_00e: NOP   0;
      A     L 80.0;
      JNB   _00f;
      L     #in_i_NoOfDataSets;
      L     2;
      +I;
      T     #tmp_i_NoOfDataSets;
_00f: NOP   0;
      A     L 80.0;
      JNB   _010;
      L     #dataSets;
      L     2;
      +I;
      T     #tmp_i_NoOfDataSets;
_010: NOP   0;
NETWORK
TITLE =
      A     #ON;
      AN    #in_b_release;
      JC    ende;
NETWORK
TITLE = move data block number to temp area (doesn't work otherwise)
//doesn't work otherwise
      L     #in_i_DBNo;
      T     #tmp_i_DBNo;
      NOP   0;
NETWORK
TITLE = open DB
      OPN   DB [#tmp_i_DBNo];
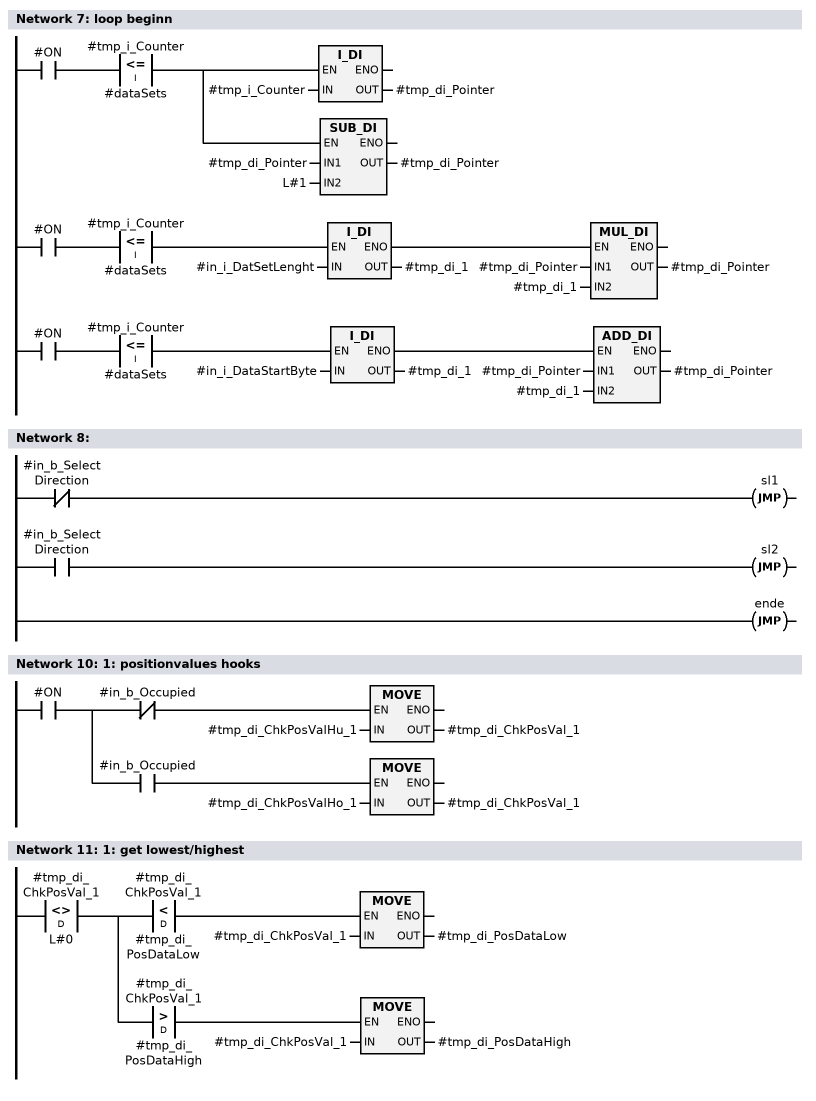
NETWORK
TITLE = loop beginn
//calculate pointer to positionvalue
scbr: A     #ON;
      A(;
      L     #tmp_i_Counter;
      L     #dataSets;
      <=I;
      );
      =     L 80.0;
      A     L 80.0;
      JNB   _011;
      L     #tmp_i_Counter;
      ITD;
      T     #tmp_di_Pointer;
_011: NOP   0;
      A     L 80.0;
      JNB   _012;
      L     #tmp_di_Pointer;
      L     L#1;
      -D;
      T     #tmp_di_Pointer;
_012: NOP   0;
      A(;
      A     L 80.0;
      JNB   _013;
      L     #in_i_DatSetLenght;
      ITD;
      T     #tmp_di_1;
      SET;
      SAVE;
      CLR;
_013: A     BR;
      );
      JNB   _014;
      L     #tmp_di_Pointer;
      L     #tmp_di_1;
      *D;
      T     #tmp_di_Pointer;
_014: NOP   0;
      A(;
      A     L 80.0;
      JNB   _015;
      L     #in_i_DataStartByte;
      ITD;
      T     #tmp_di_1;
      SET;
      SAVE;
      CLR;
_015: A     BR;
      );
      JNB   _016;
      L     #tmp_di_Pointer;
      L     #tmp_di_1;
      +D;
      T     #tmp_di_Pointer;
_016: NOP   0;
NETWORK
TITLE =
      AN    #in_b_SelectDirection;
      JC    sl1;
      A     #in_b_SelectDirection;
      JC    sl2;
      NOP   0;
      JU    ende;
NETWORK
TITLE = 1: get values from db-hooks
sl1:  NOP   0;
      L     #tmp_di_Pointer;	// load pointer
      SLD   3;	// shift left 3 bits to achieve pointer format
      LAR1;	// load adressregister 1 with pointer
      L     DBD [AR1,P#0.0];	// load position from DataBlock
      T     #tmp_di_ChkPosValHo_1;	// Transfer to temp for window check
      L     DBD [AR1,P#4.0];
      +D;
      T     #tmp_di_ChkPosValHu_1;
NETWORK
TITLE = 1: positionvalues hooks
      A     #ON;
      =     L 80.0;
      A     L 80.0;
      AN    #in_b_Occupied;
      JNB   _017;
      L     #tmp_di_ChkPosValHu_1;
      T     #tmp_di_ChkPosVal_1;
_017: NOP   0;
      A     L 80.0;
      A     #in_b_Occupied;
      JNB   _018;
      L     #tmp_di_ChkPosValHo_1;
      T     #tmp_di_ChkPosVal_1;
_018: NOP   0;
NETWORK
TITLE = 1: get lowest/highest
      L     #tmp_di_ChkPosVal_1;
      L     L#0;
      <>D;
      =     L 80.0;
      A     L 80.0;
      A(;
      L     #tmp_di_ChkPosVal_1;
      L     #tmp_di_PosDataLow;
      <D;
      );
      JNB   _019;
      L     #tmp_di_ChkPosVal_1;
      T     #tmp_di_PosDataLow;
_019: NOP   0;
      A     L 80.0;
      A(;
      L     #tmp_di_ChkPosVal_1;
      L     #tmp_di_PosDataHigh;
      >D;
      );
      JNB   _01a;
      L     #tmp_di_ChkPosVal_1;
      T     #tmp_di_PosDataHigh;
_01a: NOP   0;
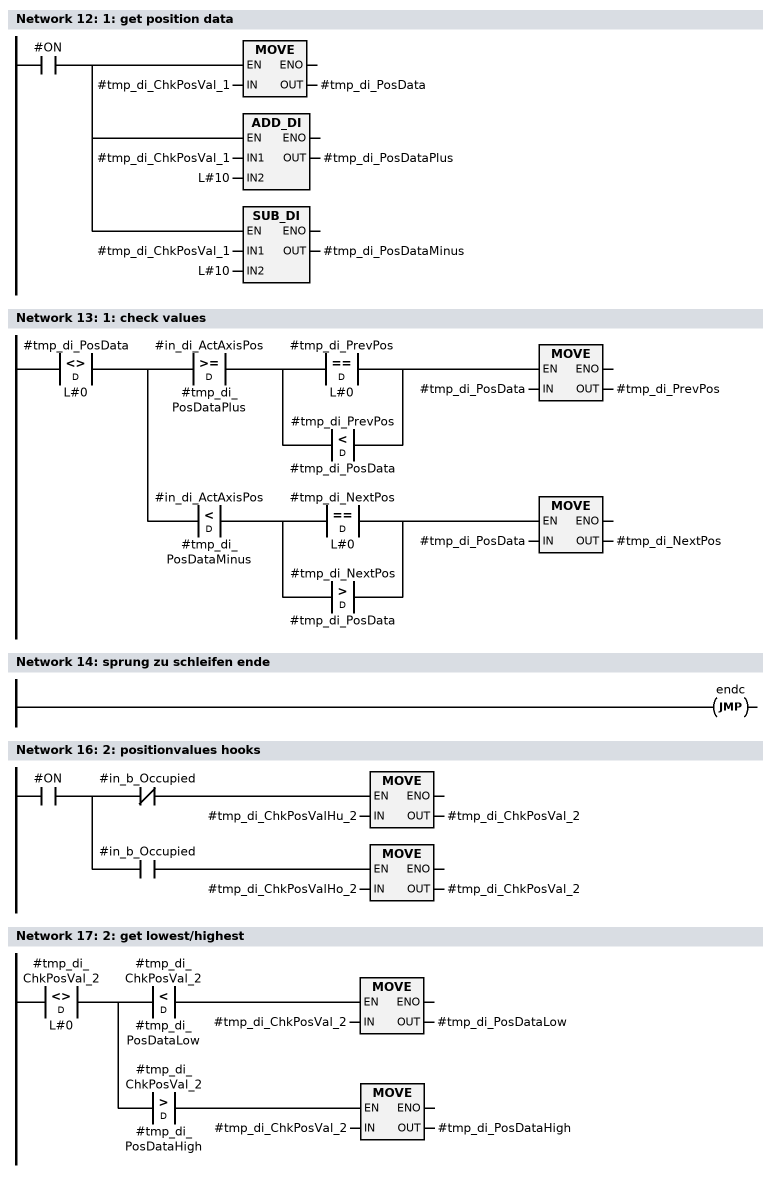
NETWORK
TITLE = 1: get position data
      A     #ON;
      =     L 80.0;
      A     L 80.0;
      JNB   _01b;
      L     #tmp_di_ChkPosVal_1;
      T     #tmp_di_PosData;
_01b: NOP   0;
      A     L 80.0;
      JNB   _01c;
      L     #tmp_di_ChkPosVal_1;
      L     L#10;
      +D;
      T     #tmp_di_PosDataPlus;
_01c: NOP   0;
      A     L 80.0;
      JNB   _01d;
      L     #tmp_di_ChkPosVal_1;
      L     L#10;
      -D;
      T     #tmp_di_PosDataMinus;
_01d: NOP   0;
NETWORK
TITLE = 1: check values
      L     #tmp_di_PosData;
      L     L#0;
      <>D;
      =     L 80.0;
      A     L 80.0;
      A(;
      L     #in_di_ActAxisPos;
      L     #tmp_di_PosDataPlus;
      >=D;
      );
      A(;
      O(;
      L     #tmp_di_PrevPos;
      L     L#0;
      ==D;
      );
      O(;
      L     #tmp_di_PrevPos;
      L     #tmp_di_PosData;
      <D;
      );
      );
      JNB   _01e;
      L     #tmp_di_PosData;
      T     #tmp_di_PrevPos;
_01e: NOP   0;
      A     L 80.0;
      A(;
      L     #in_di_ActAxisPos;
      L     #tmp_di_PosDataMinus;
      <D;
      );
      A(;
      O(;
      L     #tmp_di_NextPos;
      L     L#0;
      ==D;
      );
      O(;
      L     #tmp_di_NextPos;
      L     #tmp_di_PosData;
      >D;
      );
      );
      JNB   _01f;
      L     #tmp_di_PosData;
      T     #tmp_di_NextPos;
_01f: NOP   0;
NETWORK
TITLE = sprung zu schleifen ende
      JU    endc;
NETWORK
TITLE = 2: get values from db-hooks
sl2:  NOP   0;
      L     #tmp_di_Pointer;	// load pointer
      SLD   3;	// shift left 3 bits to achieve pointer format
      LAR1;	// load adressregister 1 with pointer
      L     DBD [AR1,P#0.0];	// load position from DataBlock
      T     #tmp_di_ChkPosValHo_2;	// Transfer to temp for window check
      L     DBD [AR1,P#4.0];
      +D;
      T     #tmp_di_ChkPosValHu_2;
NETWORK
TITLE = 2: positionvalues hooks
      A     #ON;
      =     L 80.0;
      A     L 80.0;
      AN    #in_b_Occupied;
      JNB   _020;
      L     #tmp_di_ChkPosValHu_2;
      T     #tmp_di_ChkPosVal_2;
_020: NOP   0;
      A     L 80.0;
      A     #in_b_Occupied;
      JNB   _021;
      L     #tmp_di_ChkPosValHo_2;
      T     #tmp_di_ChkPosVal_2;
_021: NOP   0;
NETWORK
TITLE = 2: get lowest/highest
      L     #tmp_di_ChkPosVal_2;
      L     L#0;
      <>D;
      =     L 80.0;
      A     L 80.0;
      A(;
      L     #tmp_di_ChkPosVal_2;
      L     #tmp_di_PosDataLow;
      <D;
      );
      JNB   _022;
      L     #tmp_di_ChkPosVal_2;
      T     #tmp_di_PosDataLow;
_022: NOP   0;
      A     L 80.0;
      A(;
      L     #tmp_di_ChkPosVal_2;
      L     #tmp_di_PosDataHigh;
      >D;
      );
      JNB   _023;
      L     #tmp_di_ChkPosVal_2;
      T     #tmp_di_PosDataHigh;
_023: NOP   0;
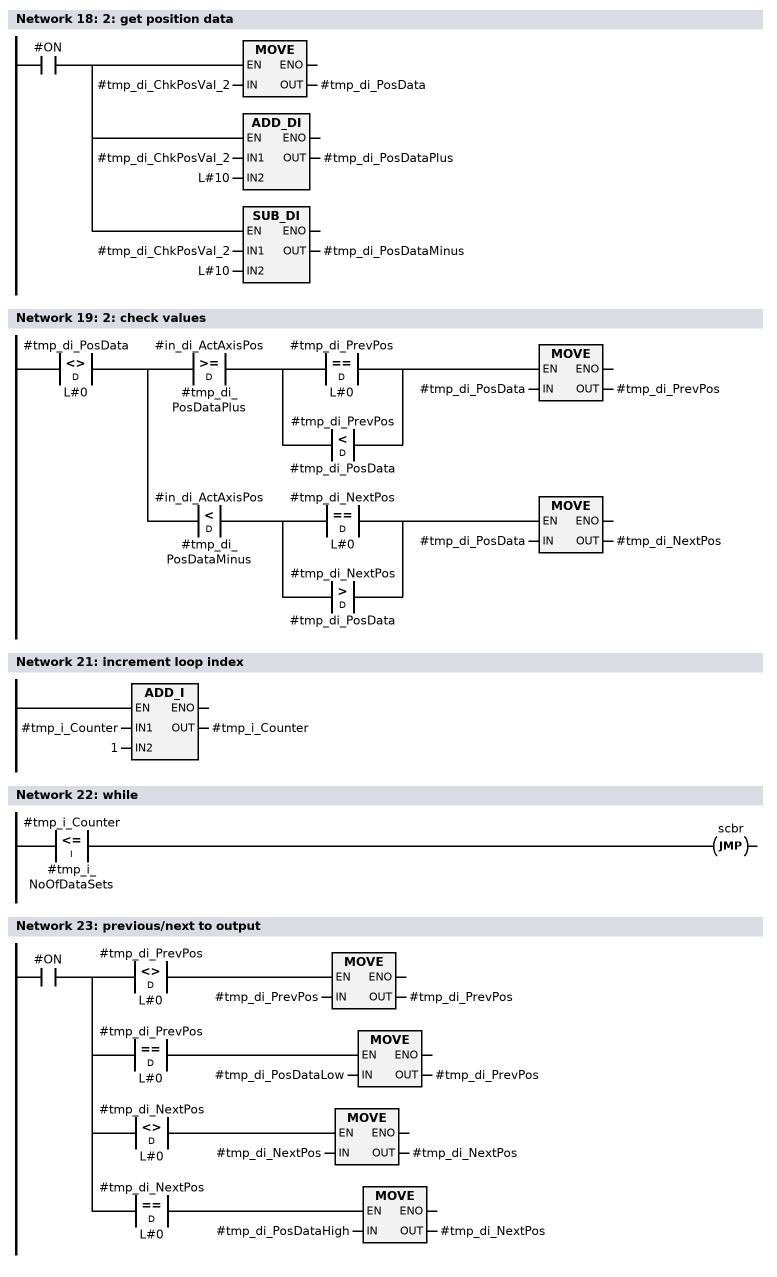
NETWORK
TITLE = 2: get position data
      A     #ON;
      =     L 80.0;
      A     L 80.0;
      JNB   _024;
      L     #tmp_di_ChkPosVal_2;
      T     #tmp_di_PosData;
_024: NOP   0;
      A     L 80.0;
      JNB   _025;
      L     #tmp_di_ChkPosVal_2;
      L     L#10;
      +D;
      T     #tmp_di_PosDataPlus;
_025: NOP   0;
      A     L 80.0;
      JNB   _026;
      L     #tmp_di_ChkPosVal_2;
      L     L#10;
      -D;
      T     #tmp_di_PosDataMinus;
_026: NOP   0;
NETWORK
TITLE = 2: check values
      L     #tmp_di_PosData;
      L     L#0;
      <>D;
      =     L 80.0;
      A     L 80.0;
      A(;
      L     #in_di_ActAxisPos;
      L     #tmp_di_PosDataPlus;
      >=D;
      );
      A(;
      O(;
      L     #tmp_di_PrevPos;
      L     L#0;
      ==D;
      );
      O(;
      L     #tmp_di_PrevPos;
      L     #tmp_di_PosData;
      <D;
      );
      );
      JNB   _027;
      L     #tmp_di_PosData;
      T     #tmp_di_PrevPos;
_027: NOP   0;
      A     L 80.0;
      A(;
      L     #in_di_ActAxisPos;
      L     #tmp_di_PosDataMinus;
      <D;
      );
      A(;
      O(;
      L     #tmp_di_NextPos;
      L     L#0;
      ==D;
      );
      O(;
      L     #tmp_di_NextPos;
      L     #tmp_di_PosData;
      >D;
      );
      );
      JNB   _028;
      L     #tmp_di_PosData;
      T     #tmp_di_NextPos;
_028: NOP   0;
NETWORK
TITLE =
endc: NOP   0;
NETWORK
TITLE = increment loop index
      L     #tmp_i_Counter;
      L     1;
      +I;
      T     #tmp_i_Counter;
      NOP   0;
NETWORK
TITLE = while 
      L     #tmp_i_Counter;
      L     #tmp_i_NoOfDataSets;
      <=I;
      JC    scbr;
NETWORK
TITLE = previous/next to output
      A     #ON;
      =     L 80.0;
      A     L 80.0;
      A(;
      L     #tmp_di_PrevPos;
      L     L#0;
      <>D;
      );
      JNB   _029;
      L     #tmp_di_PrevPos;
      T     #tmp_di_PrevPos;
_029: NOP   0;
      A     L 80.0;
      A(;
      L     #tmp_di_PrevPos;
      L     L#0;
      ==D;
      );
      JNB   _02a;
      L     #tmp_di_PosDataLow;
      T     #tmp_di_PrevPos;
_02a: NOP   0;
      A     L 80.0;
      A(;
      L     #tmp_di_NextPos;
      L     L#0;
      <>D;
      );
      JNB   _02b;
      L     #tmp_di_NextPos;
      T     #tmp_di_NextPos;
_02b: NOP   0;
      A     L 80.0;
      A(;
      L     #tmp_di_NextPos;
      L     L#0;
      ==D;
      );
      JNB   _02c;
      L     #tmp_di_PosDataHigh;
      T     #tmp_di_NextPos;
_02c: NOP   0;
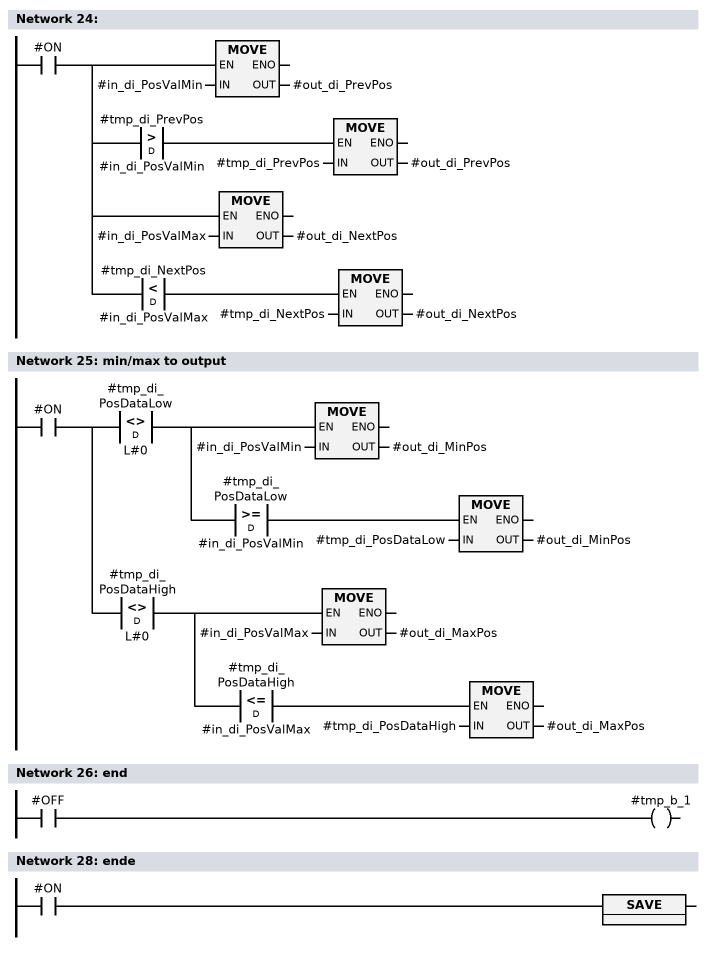
NETWORK
TITLE =
      A     #ON;
      =     L 80.0;
      A     L 80.0;
      JNB   _02d;
      L     #in_di_PosValMin;
      T     #out_di_PrevPos;
_02d: NOP   0;
      A     L 80.0;
      A(;
      L     #tmp_di_PrevPos;
      L     #in_di_PosValMin;
      >D;
      );
      JNB   _02e;
      L     #tmp_di_PrevPos;
      T     #out_di_PrevPos;
_02e: NOP   0;
      A     L 80.0;
      JNB   _02f;
      L     #in_di_PosValMax;
      T     #out_di_NextPos;
_02f: NOP   0;
      A     L 80.0;
      A(;
      L     #tmp_di_NextPos;
      L     #in_di_PosValMax;
      <D;
      );
      JNB   _030;
      L     #tmp_di_NextPos;
      T     #out_di_NextPos;
_030: NOP   0;
NETWORK
TITLE = min/max to output
      A     #ON;
      =     L 80.0;
      A     L 80.0;
      A(;
      L     #tmp_di_PosDataLow;
      L     L#0;
      <>D;
      );
      =     L 80.1;
      A     L 80.1;
      JNB   _031;
      L     #in_di_PosValMin;
      T     #out_di_MinPos;
_031: NOP   0;
      A     L 80.1;
      A(;
      L     #tmp_di_PosDataLow;
      L     #in_di_PosValMin;
      >=D;
      );
      JNB   _032;
      L     #tmp_di_PosDataLow;
      T     #out_di_MinPos;
_032: NOP   0;
      A     L 80.0;
      A(;
      L     #tmp_di_PosDataHigh;
      L     L#0;
      <>D;
      );
      =     L 80.1;
      A     L 80.1;
      JNB   _033;
      L     #in_di_PosValMax;
      T     #out_di_MaxPos;
_033: NOP   0;
      A     L 80.1;
      A(;
      L     #tmp_di_PosDataHigh;
      L     #in_di_PosValMax;
      <=D;
      );
      JNB   _034;
      L     #tmp_di_PosDataHigh;
      T     #out_di_MaxPos;
_034: NOP   0;
NETWORK
TITLE = end
ende: A     #OFF;
      =     #tmp_b_1;
NETWORK
TITLE = restore register
      LAR1  #Save_AR1;
      LAR2  #Save_AR2;
NETWORK
TITLE = ende
      A     #ON;
      SAVE;
END_FUNCTION

FUNCTION "TROGetPosVal" : VOID	// FC 1071
AUTHOR : Koenig
VERSION : 0.1
VAR_INPUT
  in_x_Enable : BOOL ;
  in_i_BrPosNo : INT ;
  in_i_TrPosNo : INT ;
  in_di_CAR1_Pos : DINT ;
  in_di_CAR2_Pos : DINT ;
END_VAR
VAR_OUTPUT
  di_TrPosVal : DINT ;
  i_DBno : INT ;
END_VAR
VAR_TEMP
  Save_AR1 : DWORD ;
  Save_AR2 : DWORD ;
  tmp_di_Pointer : DINT ;
  tmp_i : INT ;
  ON : BOOL ;
  tmp_x_OK : BOOL ;
END_VAR
BEGIN
NETWORK
TITLE = save register
      TAR1  #Save_AR1;
      TAR2  #Save_AR2;
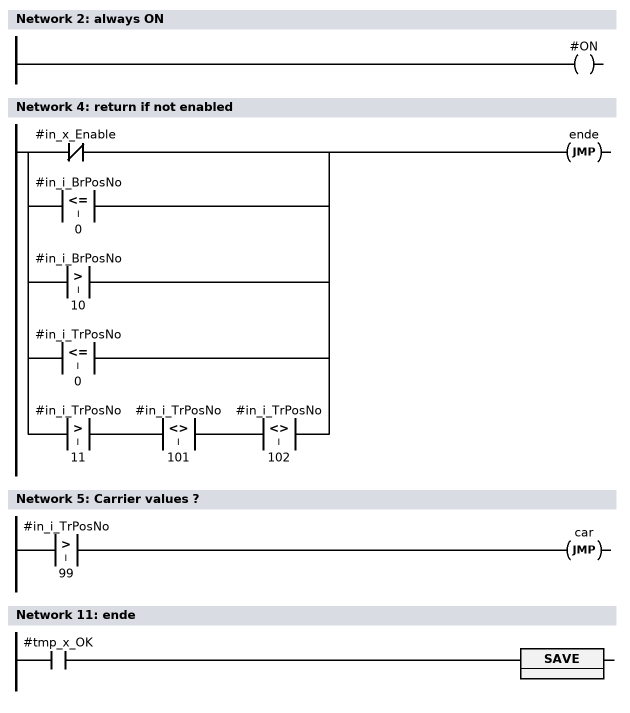
NETWORK
TITLE = always ON
      SET;
      =     #ON;
NETWORK
TITLE = init
      L     L#0;
      T     #tmp_di_Pointer;
      T     #di_TrPosVal;
      T     #i_DBno;
      CLR;
      R     #tmp_x_OK;
NETWORK
TITLE = return if not enabled
      ON    #in_x_Enable;
      O(;
      L     #in_i_BrPosNo;
      L     0;
      <=I;
      );
      O(;
      L     #in_i_BrPosNo;
      L     10;
      >I;
      );
      O(;
      L     #in_i_TrPosNo;
      L     0;
      <=I;
      );
      O;
      A(;
      L     #in_i_TrPosNo;
      L     11;
      >I;
      );
      A(;
      L     #in_i_TrPosNo;
      L     101;
      <>I;
      );
      A(;
      L     #in_i_TrPosNo;
      L     102;
      <>I;
      );
      JC    ende;
NETWORK
TITLE = Carrier values ?
      L     #in_i_TrPosNo;
      L     99;
      >I;
      JC    car;
NETWORK
TITLE = calc db no.
      L     #in_i_BrPosNo;
      L     1;
      -I;
      L     11;
      *I;
      L     #in_i_TrPosNo;
      +I;
      L     200;	// 201 is first DB
      +I;
      T     #i_DBno;
NETWORK
TITLE = get trolley value
      OPN   "TRO_Positions";
      L     L#0;
      L     #in_i_BrPosNo;
      L     1;
      -I;
      L     44;	// 11*4
      *I;
      T     #tmp_i;
      L     #in_i_TrPosNo;
      L     1;
      -I;
      L     4;
      *I;
      L     #tmp_i;
      +I;
      SLD   3;
      LAR1;
      L     DBD [AR1,P#0.0];
      T     #di_TrPosVal;
      SET;
      S     #tmp_x_OK;
      JU    ende;
NETWORK
TITLE = get carrier value
car:  NOP   0;
      L     #in_i_TrPosNo;
      L     101;
      ==I;
      JCN   c2;
      L     #in_di_CAR1_Pos;
      T     #di_TrPosVal;
      SET;
      S     #tmp_x_OK;
      JU    ende;
c2:   L     #in_i_TrPosNo;
      L     102;
      ==I;
      JCN   ende;
      L     #in_di_CAR2_Pos;
      T     #di_TrPosVal;
      SET;
      S     #tmp_x_OK;
      JU    ende;
NETWORK
TITLE = ende
ende: NOP   0;
NETWORK
TITLE = restore register
      LAR1  #Save_AR1;
      LAR2  #Save_AR2;
NETWORK
TITLE = ende
      A     #tmp_x_OK;
      SAVE;
END_FUNCTION

FUNCTION FC 1201 : VOID
VERSION : 0.0
VAR_INPUT
  Ii_Array_Pos : INT ;	//Number of the Array position
END_VAR
VAR_OUTPUT
  Od_Pos_BRI : DINT ;	//Position for the Bridge
  Od_Pos_TRO : DINT ;	//Position for the Bridge
END_VAR
VAR_TEMP
  I_COUNTER : INT ;
END_VAR
BEGIN
// body was compiled from an SCL source; compiled code not shown
END_FUNCTION

// DB 1: know-how protected block, not included

DATA_BLOCK "DB_TRO"	// DB 2
VERSION : 0.1
  STRUCT
   _di : STRUCT
    MotorTargPos : DINT ;
    MotorActPos : DINT ;
    SwsMin : DINT ;
    SwsMax : DINT ;
    PresetPos : DINT ;
    PresetData : DINT ;
    AreaWin : DINT ;
    PosWin : DINT ;
    _08 : DINT ;
    _09 : DINT ;
    _10 : DINT ;
    _11 : DINT ;
    _12 : DINT ;
    _13 : DINT ;
    _14 : DINT ;
    _15 : DINT ;
    _16 : DINT ;
    _17 : DINT ;
    _18 : DINT ;
    Offset : DINT ;
    ManPrevPos : DINT ;
    ManActPos : DINT ;
    ManNextPos : DINT ;
    ManMinPos : DINT ;
    ManMaxPos : DINT ;
    ManTargPosVal : DINT ;
    _26 : DINT ;
    _27 : DINT ;
    _28 : DINT ;
    _29 : DINT ;
    _30 : DINT ;
    _31 : DINT ;
    _32 : DINT ;
    _33 : DINT ;
    _34 : DINT ;
    ActPosMinusOffset : DINT ;
    TargPosPlusOffset : DINT ;
    _37 : DINT ;
    _38 : DINT ;
    _39 : DINT ;
    _40 : DINT ;
    _41 : DINT ;
    _42 : DINT ;
    _43 : DINT ;
    _44 : DINT ;
    _45 : DINT ;
    _46 : DINT ;
    _47 : DINT ;
    _48 : DINT ;
    _49 : DINT ;
    _50 : DINT ;
    _51 : DINT ;
    _52 : DINT ;
    _53 : DINT ;
    _54 : DINT ;
    _55 : DINT ;
    _56 : DINT ;
    _57 : DINT ;
    _58 : DINT ;
    _59 : DINT ;
    _60 : DINT ;
    _61 : DINT ;
    _62 : DINT ;
    _63 : DINT ;
    _64 : DINT ;
    _65 : DINT ;
    _66 : DINT ;
    _67 : DINT ;
    _68 : DINT ;
    _69 : DINT ;
    _70 : DINT ;
    _71 : DINT ;
    _72 : DINT ;
    _73 : DINT ;
    _74 : DINT ;
   END_STRUCT ;
   _i : STRUCT
    MotorIn_00 : INT ;
    MotorIn_01 : INT ;
    MotorIn_02 : INT ;
    MotorIn_03 : INT ;
    MotorIn_04 : INT ;
    MotorIn_05 : INT ;
    MotorOut_00 : INT ;
    MotorOut_01 : INT ;
    MotorOut_02 : INT ;
    MotorOut_03 : INT ;
    MotorOut_04 : INT ;
    MotorOut_05 : INT ;
    MotorCrtWord : INT ;
    MotorTargSpeed : INT ;
    MotorTargAcc : INT ;
    MotorTargDeacc : INT ;
    MotorStateWord : INT ;
    MotorActSpeed : INT ;
    MotorActCurrent : INT ;
    MotorActWorkLoad : INT ;
    SourcePosNo : INT ;
    TargPosNo : INT ;
    ActAreaNo : INT ;
    ServiceV : INT ;
    ManualV : INT ;
    OnlineV : INT ;
    ForcedSlowV : INT ;
    RuntimeSec : INT ;
    ActPosNo : INT ;
    ScanAreaNo : INT ;
    SpeedManual : INT ;
    SafetySpeed : INT ;	//sichere Geschwindigkeit (1/min)
    SpeedForcSlow : INT ;
    SpeedManSlo : INT ;
    Acceleration : INT ;
    Deacceleration : INT ;
    _36 : INT ;
    ManTargPosNo : INT ;
    PrevPosNo : INT ;
    NextPosNo : INT ;
    MinPosNo : INT ;
    MaxPosNo : INT ;
    _42 : INT ;
    _43 : INT ;
    _44 : INT ;
    ActLIF_DBNo : INT ;
    _46 : INT ;
    _47 : INT ;
    _48 : INT ;
    _49 : INT ;
    _50 : INT ;
    _51 : INT ;
    _52 : INT ;
    _53 : INT ;
    _54 : INT ;
    _55 : INT ;
    _56 : INT ;
    _57 : INT ;
    _58 : INT ;
    _59 : INT ;
    _60 : INT ;
    _61 : INT ;
    _62 : INT ;
    _63 : INT ;
    _64 : INT ;
    _65 : INT ;
    _66 : INT ;
    _67 : INT ;
    _68 : INT ;
    _69 : INT ;
    _70 : INT ;
    _71 : INT ;
    _72 : INT ;
    _73 : INT ;
    _74 : INT ;
    _75 : INT ;
    _76 : INT ;
    _77 : INT ;
    _78 : INT ;
    _79 : INT ;
    _80 : INT ;
    _81 : INT ;
    _82 : INT ;
    _83 : INT ;
    _84 : INT ;
    _85 : INT ;
    _86 : INT ;
    _87 : INT ;
    _88 : INT ;
    _89 : INT ;
    _90 : INT ;
    _91 : INT ;
    _92 : INT ;
    _93 : INT ;
    _94 : INT ;
    _95 : INT ;
    _96 : INT ;
    _97 : INT ;
    _98 : INT ;
    DriveErrorCode : INT ;
   END_STRUCT ;
   _x : STRUCT
    InchMinus : BOOL ;
    InchPlus : BOOL ;
    TargIsPos : BOOL ;
    RelForPos : BOOL ;
    MovesMinus : BOOL ;
    MovesPlus : BOOL ;
    Moves : BOOL ;
    InArea : BOOL ;
    InPos : BOOL ;
    FastStop : BOOL ;
    ManPosFound : BOOL ;
    MotorReady : BOOL ;
    MotorRefOk : BOOL ;
    ForcedSlow : BOOL ;
    StartPos : BOOL ;
    Position_Found : BOOL ;
    _16 : BOOL ;
    _17 : BOOL ;
    DelayFaststop : BOOL ;
    ReleaseScan : BOOL ;
    ScanInPos : BOOL ;
    AutoInPos : BOOL ;
    TargPosFront : BOOL ;
    TargPosBack : BOOL ;
    InPosCart : BOOL ;
    _25 : BOOL ;
    _26 : BOOL ;
    _27 : BOOL ;
    _28 : BOOL ;
    _29 : BOOL ;
    _30 : BOOL ;
    _31 : BOOL ;
    _32 : BOOL ;
    _33 : BOOL ;
    _34 : BOOL ;
    _35 : BOOL ;
    _36 : BOOL ;
    _37 : BOOL ;
    _38 : BOOL ;
    _39 : BOOL ;
    _40 : BOOL ;
    _41 : BOOL ;
    _42 : BOOL ;
    _43 : BOOL ;
    _44 : BOOL ;
    _45 : BOOL ;
    _46 : BOOL ;
    _47 : BOOL ;
    _48 : BOOL ;
    _49 : BOOL ;
    _50 : BOOL ;
    PresetOffset : BOOL ;
    _52 : BOOL ;
    _53 : BOOL ;
    _54 : BOOL ;
    _55 : BOOL ;
    _56 : BOOL ;
    _57 : BOOL ;
    _58 : BOOL ;
    _59 : BOOL ;
    _60 : BOOL ;
    _61 : BOOL ;
    fs_Minus_SW : BOOL ;	//forced slow software
    fs_Plus_Sw : BOOL ;	//forced slow software
    _64 : BOOL ;
    _65 : BOOL ;
    _66 : BOOL ;
    _67 : BOOL ;
    _68 : BOOL ;
    _69 : BOOL ;
    _70 : BOOL ;
    _71 : BOOL ;
    _72 : BOOL ;
    _73 : BOOL ;
    _74 : BOOL ;
    _75 : BOOL ;
    _76 : BOOL ;
    _77 : BOOL ;
    _78 : BOOL ;
    _79 : BOOL ;
    _80 : BOOL ;
    _81 : BOOL ;
    _82 : BOOL ;
    _83 : BOOL ;
    _84 : BOOL ;
    _85 : BOOL ;
    _86 : BOOL ;
    _87 : BOOL ;
    _88 : BOOL ;
    _89 : BOOL ;
    _90 : BOOL ;
    _91 : BOOL ;
    _92 : BOOL ;
    _93 : BOOL ;
    _94 : BOOL ;
    _95 : BOOL ;
   END_STRUCT ;
  END_STRUCT ;	
BEGIN
   _di.MotorTargPos := L#160212;
   _di.MotorActPos := L#160213;
   _di.SwsMin := L#1980;
   _di.SwsMax := L#390000;
   _di.AreaWin := L#10;
   _di.PosWin := L#1;
   _di.ManPrevPos := L#5134;
   _di.ManActPos := L#7046;
   _di.ManNextPos := L#9344;
   _di.ManMinPos := L#1313;
   _di.ManMaxPos := L#9344;
   _di.ManTargPosVal := L#3223;
   _di.ActPosMinusOffset := L#160213;
   _di.TargPosPlusOffset := L#160212;
   _di._45 := L#-184;
   _i.MotorOut_00 := 2048;
   _i.MotorOut_03 := 12;
   _i.MotorOut_04 := 4000;
   _i.MotorOut_05 := 4000;
   _i.MotorCrtWord := 6144;
   _i.MotorTargSpeed := 300;
   _i.MotorTargAcc := 150;
   _i.MotorTargDeacc := 150;
   _i.MotorStateWord := 518;
   _i.TargPosNo := 8;
   _i.ActAreaNo := 4;
   _i.ServiceV := 1;
   _i.ManualV := 30;
   _i.OnlineV := 100;
   _i.ForcedSlowV := 5;
   _i.ActPosNo := 99;
   _i.ScanAreaNo := 8;
   _i.SpeedManual := 2;
   _i.SpeedForcSlow := 5;
   _i.SpeedManSlo := 2;
   _i.Acceleration := 3000;
   _i.Deacceleration := 3000;
   _i._36 := 2;
   _i.ManTargPosNo := 2;
   _i.PrevPosNo := 3;
   _i.NextPosNo := 5;
   _i.MinPosNo := 1;
   _i.MaxPosNo := 5;
   _i.ActLIF_DBNo := 201;
   _i.DriveErrorCode := 2;
   _x.InArea := TRUE;
   _x.FastStop := TRUE;
   _x.MotorReady := TRUE;
   _x.MotorRefOk := TRUE;
   _x.ScanInPos := TRUE;
   _x.AutoInPos := TRUE;
   _x._56 := TRUE;
END_DATA_BLOCK

DATA_BLOCK "DB_LIF"	// DB 3
VERSION : 0.1
  STRUCT
   _di : STRUCT
    MotorTargPos : DINT ;
    MotorActPos : DINT ;
    SwsMin : DINT ;
    SwsMax : DINT ;
    PresetPos : DINT ;
    PresetData : DINT ;
    AreaWin : DINT ;
    PosWin : DINT ;
    PointerDataset : DINT ;
    ValPosTop : DINT ;
    ValPosIntHo : DINT ;
    ValOffsetIntHu : DINT ;
    ValPosWanne : DINT ;
    ValPosTurnHo : DINT ;
    ValPosTurnHu : DINT ;
    ValPosHoAct : DINT ;
    ValPosHuAct : DINT ;
    ValPosSwitchPointCarts : DINT ;
    ValPosSwitchPointTurn : DINT ;
    OffsetLift : DINT ;
    ManPrevPos : DINT ;
    ManActPos : DINT ;
    ManNextPos : DINT ;
    ManMinPos : DINT ;
    ManMaxPos : DINT ;
    ManTargPos : DINT ;
    ValSafetyAreaWama : DINT ;
    AreaCartToHighMin : DINT ;
    AreaCartToHighMax : DINT ;
    AreaCoverMin : DINT ;
    AreaCoverMax : DINT ;
    ValToWid_3 : DINT ;
    _32 : DINT ;
    _33 : DINT ;
    _34 : DINT ;
    ActPosMinusOffset : DINT ;
    TargPosPlusOffset : DINT ;
    _37 : DINT ;
    _38 : DINT ;
    _39 : DINT ;
    LastTelCenter : DINT ;
    MaxDistanceTel : DINT ;
    _42 : DINT ;
    _43 : DINT ;
    _44 : DINT ;
    _45 : DINT ;
    _46 : DINT ;
    _47 : DINT ;
    _48 : DINT ;
    _49 : DINT ;
    _50 : DINT ;
    _51 : DINT ;
    _52 : DINT ;
    _53 : DINT ;
    _54 : DINT ;
    _55 : DINT ;
    _56 : DINT ;
    _57 : DINT ;
    _58 : DINT ;
    _59 : DINT ;
    _60 : DINT ;
    _61 : DINT ;
    _62 : DINT ;
    _63 : DINT ;
    _64 : DINT ;
    _65 : DINT ;
    _66 : DINT ;
    _67 : DINT ;
    _68 : DINT ;
    _69 : DINT ;
    _70 : DINT ;
    _71 : DINT ;
    _72 : DINT ;
    _73 : DINT ;
    _74 : DINT ;
   END_STRUCT ;
   _i : STRUCT
    MotorIn_00 : INT ;
    MotorIn_01 : INT ;
    MotorIn_02 : INT ;
    MotorIn_03 : INT ;
    MotorIn_04 : INT ;
    MotorIn_05 : INT ;
    MotorOut_00 : INT ;
    MotorOut_01 : INT ;
    MotorOut_02 : INT ;
    MotorOut_03 : INT ;
    MotorOut_04 : INT ;
    MotorOut_05 : INT ;
    MotorCrtWord : INT ;
    MotorTargSpeed : INT ;
    MotorTargAcc : INT ;
    MotorTargDeacc : INT ;
    MotorStateWord : INT ;
    MotorActSpeed : INT ;
    MotorActCurrent : INT ;
    MotorActWorkLoad : INT ;
    SourcePosNo : INT ;
    TargPosNo : INT ;
    ActAreaNo : INT ;
    ServiceV : INT ;
    ManualV : INT ;
    OnlineV : INT ;
    ForcedSlowV : INT ;
    RuntimeSec : INT ;
    ActPosNo : INT ;
    ActLiDbNo_1 : INT ;
    SpeedManual : INT ;
    ActHooktype : INT ;
    SpeedForcSlow : INT ;
    SpeedManSlow : INT ;
    Acceleration : INT ;
    Deacceleration : INT ;
    FcErrorNo : INT ;
    ManTargPosNo : INT ;
    ActCircMax : INT ;
    ActLiDbNo_2 : INT ;
    ActLIF_DB : INT ;
    _41 : INT ;
    _42 : INT ;
    _43 : INT ;
    _44 : INT ;
    _45 : INT ;
    _46 : INT ;
    _47 : INT ;
    _48 : INT ;
    _49 : INT ;
    _50 : INT ;
    _51 : INT ;
    _52 : INT ;
    _53 : INT ;
    _54 : INT ;
    _55 : INT ;
    _56 : INT ;
    _57 : INT ;
    _58 : INT ;
    _59 : INT ;
    _60 : INT ;
    _61 : INT ;
    _62 : INT ;
    _63 : INT ;
    _64 : INT ;
    _65 : INT ;
    _66 : INT ;
    _67 : INT ;
    _68 : INT ;
    _69 : INT ;
    _70 : INT ;
    _71 : INT ;
    _72 : INT ;
    _73 : INT ;
    _74 : INT ;
    _75 : INT ;
    _76 : INT ;
    _77 : INT ;
    _78 : INT ;
    _79 : INT ;
    _80 : INT ;
    _81 : INT ;
    _82 : INT ;
    _83 : INT ;
    _84 : INT ;
    _85 : INT ;
    _86 : INT ;
    _87 : INT ;
    _88 : INT ;
    _89 : INT ;
    _90 : INT ;
    _91 : INT ;
    _92 : INT ;
    _93 : INT ;
    _94 : INT ;
    _95 : INT ;
    _96 : INT ;
    _97 : INT ;
    _98 : INT ;
    DriveErrorCode : INT ;
   END_STRUCT ;
   _x : STRUCT
    InchMinus : BOOL ;
    InchPlus : BOOL ;
    TargIsPos : BOOL ;
    RelForPos : BOOL ;
    MovesMinus : BOOL ;
    MovesPlus : BOOL ;
    Moves : BOOL ;
    InArea : BOOL ;
    InPos : BOOL ;
    FastStop : BOOL ;
    ManPosFound : BOOL ;
    MotorReady : BOOL ;
    MotorRefOk : BOOL ;
    ForcedSlow : BOOL ;
    StartPos : BOOL ;
    InPosHookover : BOOL ;
    InPosHookunder : BOOL ;
    InPosTop : BOOL ;
    DelayFaststop : BOOL ;
    ReleaseScan : BOOL ;
    ScanInPos : BOOL ;
    AutoInPos : BOOL ;
    TargIsTop : BOOL ;
    TargIsIntPos : BOOL ;
    InAreaTop : BOOL ;
    PosTop : BOOL ;
    InAreaIntPos : BOOL ;
    InIntPosHo : BOOL ;
    InIntPosHu : BOOL ;
    RequireClamp : BOOL ;
    TargIsHookover : BOOL ;
    TargIsHookunder : BOOL ;
    LiClamped : BOOL ;
    LiDeclamped : BOOL ;
    ReleasePlus : BOOL ;
    ReleaseMinus : BOOL ;
    SensorsOn : BOOL ;
    IntPosOccup : BOOL ;
    WanneOk : BOOL ;
    InHookArea : BOOL ;
    Lock_Rack : BOOL ;
    Lock_Carts : BOOL ;
    Lock_Washer : BOOL ;
    Lock_TurnTable : BOOL ;
    Lock_Pallets : BOOL ;
    Lock_WashPlaces : BOOL ;
    Lock_internal : BOOL ;
    Lock_Lift : BOOL ;
    PreStartPos : BOOL ;
    HelpBuffer : BOOL ;
    StopAtBuffer : BOOL ;
    PresetOffset : BOOL ;
    CopyLiftDataOK : BOOL ;
    ChkCableDrum1 : BOOL ;
    ChkCableDrum2 : BOOL ;
    CopyDBOrder : BOOL ;
    InSafetyAreaWAMA : BOOL ;
    TargIsSafety : BOOL ;
    InSafetyPosWAMA : BOOL ;
    InPosSwitchPoint : BOOL ;
    TargetSwitchPoint : BOOL ;
    InAreaSwitchPoint : BOOL ;
    fs_Minus_SW : BOOL ;
    fs_Plus_SW : BOOL ;
    TopPosFound : BOOL ;
    TargIsLowest : BOOL ;
    ReleaseWidth1 : BOOL ;
    Dir_1 : BOOL ;
    Dir_2 : BOOL ;
    LiftInAreaLS1 : BOOL ;
    SelectDirectionFront : BOOL ;
    DbCopyOk_Scan : BOOL ;
    ScanInTopPosition : BOOL ;
    TopPosStop : BOOL ;
    LiftInAreaLS2 : BOOL ;
    LiftInAreaLS3 : BOOL ;
    _76 : BOOL ;
    _77 : BOOL ;
    DBCopyBusy_Auto : BOOL ;
    DbCopyOk_Auto : BOOL ;
    _80 : BOOL ;
    DBCopyBusy_Scan : BOOL ;
    _82 : BOOL ;
    _83 : BOOL ;
    _84 : BOOL ;
    _85 : BOOL ;
    _86 : BOOL ;
    _87 : BOOL ;
    _88 : BOOL ;
    _89 : BOOL ;
    _90 : BOOL ;
    _91 : BOOL ;
    _92 : BOOL ;
    _93 : BOOL ;
    _94 : BOOL ;
    _95 : BOOL ;
   END_STRUCT ;
  END_STRUCT ;	
BEGIN
   _di.MotorTargPos := L#5860;
   _di.MotorActPos := L#5859;
   _di.SwsMin := L#330;
   _di.SwsMax := L#7000;
   _di.AreaWin := L#150;
   _di.PosWin := L#1;
   _di.PointerDataset := L#56;
   _di.ValPosTop := L#342;
   _di.ValPosIntHo := L#337;
   _di.ValOffsetIntHu := L#60;
   _di.ValPosTurnHo := L#4030;
   _di.ValPosTurnHu := L#5069;
   _di.ValPosHoAct := L#5745;
   _di.ValPosHuAct := L#5860;
   _di.ValPosSwitchPointCarts := L#4200;
   _di.ValPosSwitchPointTurn := L#4100;
   _di.ManPrevPos := L#3750;
   _di.ManActPos := L#4000;
   _di.ManNextPos := L#4100;
   _di.ManMinPos := L#337;
   _di.ManMaxPos := L#6500;
   _di.ManTargPos := L#6316;
   _di.ValSafetyAreaWama := L#3515;
   _di.AreaCartToHighMin := L#4480;
   _di.AreaCartToHighMax := L#4525;
   _di.AreaCoverMin := L#4480;
   _di.AreaCoverMax := L#4525;
   _di.ActPosMinusOffset := L#5859;
   _di.TargPosPlusOffset := L#5860;
   _di._37 := L#204;
   _di.LastTelCenter := L#5379;
   _di.MaxDistanceTel := L#150;
   _i.MotorOut_00 := 2048;
   _i.MotorOut_02 := -17336;
   _i.MotorOut_03 := 12;
   _i.MotorOut_04 := 400;
   _i.MotorOut_05 := 400;
   _i.MotorCrtWord := 6148;
   _i.MotorTargSpeed := 50;
   _i.MotorTargAcc := 350;
   _i.MotorTargDeacc := 350;
   _i.MotorStateWord := 518;
   _i.TargPosNo := 2;
   _i.ActAreaNo := 2;
   _i.ServiceV := 3;
   _i.ManualV := 30;
   _i.OnlineV := 80;
   _i.ForcedSlowV := 4;
   _i.ActPosNo := 2;
   _i.ActLiDbNo_1 := 173;
   _i.SpeedManual := 30;
   _i.ActHooktype := 10;
   _i.SpeedForcSlow := 9;
   _i.SpeedManSlow := 3;
   _i.Acceleration := 2000;
   _i.Deacceleration := 2000;
   _i.FcErrorNo := 2;
   _i.ActCircMax := 980;
   _i.ActLiDbNo_2 := 174;
   _i.ActLIF_DB := 92;
   _i._42 := 5122;
   _i._45 := 134;
   _i.DriveErrorCode := 2;
   _x.InArea := TRUE;
   _x.FastStop := TRUE;
   _x.MotorReady := TRUE;
   _x.MotorRefOk := TRUE;
   _x.ForcedSlow := TRUE;
   _x.InPosHookunder := TRUE;
   _x.ReleaseScan := TRUE;
   _x.ScanInPos := TRUE;
   _x.AutoInPos := TRUE;
   _x.InAreaTop := TRUE;
   _x.LiClamped := TRUE;
   _x.ReleaseMinus := TRUE;
   _x.SensorsOn := TRUE;
   _x.Lock_internal := TRUE;
   _x.Lock_Lift := TRUE;
   _x.Dir_2 := TRUE;
   _x.SelectDirectionFront := TRUE;
   _x._76 := TRUE;
   _x.DbCopyOk_Auto := TRUE;
   _x.DBCopyBusy_Scan := TRUE;
END_DATA_BLOCK

DATA_BLOCK "DB_TEL"	// DB 4
VERSION : 0.1
  STRUCT
   _di : STRUCT
    MotorTargPos : DINT ;
    MotorActPos : DINT ;
    SwsMin : DINT ;
    SwsMax : DINT ;
    PresetPos : DINT ;
    PresetData : DINT ;
    AreaWin : DINT ;
    PosWin : DINT ;
    SlowWin : DINT ;
    StopWin : DINT ;
    ValPosCenter : DINT ;
    ValActPos1 : DINT ;
    ValActPos2 : DINT ;
    ValActPos3 : DINT ;
    VolPosInternHook : DINT ;
    ValueLastCycle : DINT ;
    _16 : DINT ;
    _17 : DINT ;
    _18 : DINT ;
    _19 : DINT ;
    ManPrevPos : DINT ;
    ManActPos : DINT ;
    ManNextPos : DINT ;
    ManMinPos : DINT ;
    ManMaxPos : DINT ;
    ManTargPos : DINT ;
    _26 : DINT ;
    _27 : DINT ;
    _Enco_Helpflag1 : DINT ;	//Encoder Schmiermerker größer
    _Enco_Helpflag2 : DINT ;	//Encoder Schmiermerker kleiner
    _ActEncoder_mm : DINT ;	//Istwert SSI Encoder in mm
    _PresetEncoder_mm : DINT ;	//Preset SSI Encoder (Teleskope Mittelstellung)
    _FactorEncoder : DINT ;	//Umrechungsfaktor SSI Encoder auf mm
    _Enc_Korrektur : DINT ;	//wird zur Umrechnung benoetigt (man kann nur auf 0 Preseten)
    _Enc_Window : DINT ;	//Positions Fenster
    ActPosMinusOffset : DINT ;
    TargPosPlusOffset : DINT ;
    _37 : DINT ;
    _38 : DINT ;
    _39 : DINT ;
    _Pos_Center : DINT ;	//Mitte
    _Pos_left_big : DINT ;	//links groß
    _Pos_left_mid : DINT ;	//links mittel
    _Pos_left_small_1 : DINT ;	//links klein 1
    _Pos_left_small_2 : DINT ;	//links klein 2
    _Pos_right_big : DINT ;	//rechts groß
    _Pos_right_mid : DINT ;	//rechts mittel
    _Pos_right_small_1 : DINT ;	//rechts klein 1
    _Pos_right_small_2 : DINT ;	//rechts klein 2
    _Pos_res_1 : DINT ;	//res
    _Pos_res_2 : DINT ;	//res
    _51 : DINT ;
    _52 : DINT ;
    _53 : DINT ;
    _54 : DINT ;
    _55 : DINT ;
    _56 : DINT ;
    _57 : DINT ;
    _58 : DINT ;
    _59 : DINT ;
    _60 : DINT ;
    _61 : DINT ;
    _62 : DINT ;
    _63 : DINT ;
    _64 : DINT ;
    _65 : DINT ;
    _66 : DINT ;
    _67 : DINT ;
    _68 : DINT ;
    _69 : DINT ;
    _70 : DINT ;
    _71 : DINT ;
    _72 : DINT ;
    _73 : DINT ;
    _74 : DINT ;
   END_STRUCT ;
   _i : STRUCT
    MotorIn_00 : INT ;
    MotorIn_01 : INT ;
    MotorIn_02 : INT ;
    MotorIn_03 : INT ;
    MotorIn_04 : INT ;
    MotorIn_05 : INT ;
    MotorOut_00 : INT ;
    MotorOut_01 : INT ;
    MotorOut_02 : INT ;
    MotorOut_03 : INT ;
    MotorOut_04 : INT ;
    MotorOut_05 : INT ;
    MotorCrtWord : INT ;
    MotorTargSpeed : INT ;
    MotorTargAcc : INT ;
    MotorTargDeacc : INT ;
    MotorStateWord : INT ;
    MotorActSpeed : INT ;
    MotorActCurrent : INT ;
    MotorActWorkLoad : INT ;
    SourcePosNo : INT ;
    TargPosNo : INT ;
    ActAreaNo : INT ;
    ServiceV : INT ;
    ManualV : INT ;
    OnlineV : INT ;
    ForcedSlowV : INT ;
    RuntimeSec : INT ;
    ActPosNo : INT ;
    _29 : INT ;
    ActCylTypeTelescopes : INT ;
    ActDiamterCylTelescopes : INT ;
    ActCircumCylTelescopes : INT ;
    ActValueMeasureDiameter : INT ;
    _34 : INT ;
    _35 : INT ;
    _36 : INT ;
    ManTargPosNo : INT ;
    _38 : INT ;
    _39 : INT ;
    _40 : INT ;
    _41 : INT ;
    _42 : INT ;
    _43 : INT ;
    _44 : INT ;
    EncoderErrCode : INT ;
    _46 : INT ;
    _47 : INT ;
    _48 : INT ;
    _49 : INT ;
    _50 : INT ;
    _51 : INT ;
    _52 : INT ;
    _53 : INT ;
    _54 : INT ;
    _55 : INT ;
    _56 : INT ;
    _57 : INT ;
    _58 : INT ;
    _59 : INT ;
    _60 : INT ;
    _61 : INT ;
    _62 : INT ;
    _63 : INT ;
    _64 : INT ;
    _65 : INT ;
    _66 : INT ;
    _67 : INT ;
    _68 : INT ;
    _69 : INT ;
    _70 : INT ;
    _71 : INT ;
    _72 : INT ;
    _73 : INT ;
    _74 : INT ;
    _75 : INT ;
    _76 : INT ;
    _77 : INT ;
    _78 : INT ;
    _79 : INT ;
    _80 : INT ;
    _81 : INT ;
    _82 : INT ;
    _83 : INT ;
    _84 : INT ;
    _85 : INT ;
    _86 : INT ;
    _87 : INT ;
    _88 : INT ;
    _89 : INT ;
    _90 : INT ;
    _91 : INT ;
    _92 : INT ;
    _93 : INT ;
    _94 : INT ;
    _95 : INT ;
    _96 : INT ;
    _97 : INT ;
    _98 : INT ;
    DriveErrorCode : INT ;
   END_STRUCT ;
   _x : STRUCT
    InchMinus : BOOL ;
    InchPlus : BOOL ;
    TargIsPos : BOOL ;
    RelForPos : BOOL ;
    MovesMinus : BOOL ;
    MovesPlus : BOOL ;
    Moves : BOOL ;
    InArea : BOOL ;
    InPos : BOOL ;
    FastStop : BOOL ;
    ManPosFound : BOOL ;
    MotorReady : BOOL ;
    MotorRefOk : BOOL ;
    ForcedSlow : BOOL ;
    StartPos : BOOL ;
    TargIsCenter : BOOL ;
    ReleaseToHook : BOOL ;
    InPosCenter : BOOL ;
    InAreaCenter : BOOL ;
    ReleaseScan : BOOL ;
    ScanInPos : BOOL ;
    AutoInPos : BOOL ;
    InPosIntern : BOOL ;
    TargIsInternPos : BOOL ;
    Occup : BOOL ;
    Free : BOOL ;
    TelPos1_FsOccup : BOOL ;
    TelPos2_FsOccup : BOOL ;
    TelPos3_FsOccup : BOOL ;
    TelPos1_BsOccup : BOOL ;
    TelPos2_BsOccup : BOOL ;
    TelPos3_BsOccup : BOOL ;
    AutoPosOk : BOOL ;
    BuffOccOK : BOOL ;
    ReleasePlus : BOOL ;
    ReleaseMinus : BOOL ;
    PulsRcPlus : BOOL ;
    PulsRcMinus : BOOL ;
    PosFront : BOOL ;	//left from the center
    PosRear : BOOL ;	//right from the center
    Lock01 : BOOL ;
    Lock02 : BOOL ;
    Lock03 : BOOL ;
    Lock04 : BOOL ;
    Lock05 : BOOL ;
    Lock06 : BOOL ;
    Lock07 : BOOL ;
    PosCenterChk : BOOL ;
    BuffOcc : BOOL ;
    BuffFree : BOOL ;
    PosFoundCenter : BOOL ;
    PosHookIn : BOOL ;	//Haken innen
    PosHookMid : BOOL ;	//Haken Mitte
    PosHookOut : BOOL ;	//Haken aussen
    _54 : BOOL ;
    LockSum : BOOL ;
    ScanInStopPos : BOOL ;
    FU_Off : BOOL ;	//FU stop in PosFound
    OccStateOK : BOOL ;	//beide Sensoren gleich
    Lock08 : BOOL ;
    Lock09 : BOOL ;
    Lock10 : BOOL ;
    fs_Minus_SW : BOOL ;	//forced slow software
    fs_Plus_SW : BOOL ;	//forced slow software
    pFl_TEL_Occ : BOOL ;
    nFl_TEL_Occ : BOOL ;
    ManTargetRight : BOOL ;
    HookTypePallett : BOOL ;
    _68 : BOOL ;
    _69 : BOOL ;
    OccupSteute : BOOL ;	//occupation state steute
    Free_Steute : BOOL ;	//occupation state steute
    EncoderError : BOOL ;
    Chk_Fs1Hu_after : BOOL ;
    Chk_Bs1Hu_after : BOOL ;
    Chk_Fs2Hu_after : BOOL ;
    Chk_Bs2Hu_after : BOOL ;
    Chk_Fs3Hu_after : BOOL ;
    Chk_Bs3Hu_after : BOOL ;
    Chk_Fs1Hu_before : BOOL ;
    Chk_Bs1Hu_before : BOOL ;
    Chk_Fs2Hu_before : BOOL ;
    Chk_Bs2Hu_before : BOOL ;
    Chk_Fs3Hu_before : BOOL ;
    Chk_Bs3Hu_before : BOOL ;
    Chk_Fs1Ho : BOOL ;
    Chk_Bs1Ho : BOOL ;
    Chk_Fs2Ho : BOOL ;
    Chk_Bs2Ho : BOOL ;
    Chk_Fs3Ho : BOOL ;
    Chk_Bs3Ho : BOOL ;
    Chk_Hu_OK_after : BOOL ;
    Chk_Hu_OK_before : BOOL ;
    Chk_Ho_OK : BOOL ;
    _94 : BOOL ;
    _95 : BOOL ;
    DRC_MotorErr : BOOL ;
    not_Referenced : BOOL ;
    InPosition : BOOL ;
    Ready : BOOL ;
    TargetPos : INT ;
    ActualPos : INT ;
   END_STRUCT ;
   _X_TEL_POS_Center : BOOL ;
   _X_TEL_POS_1 : BOOL ;
   _X_TEL_POS_2 : BOOL ;
   _X_TEL_POS_3 : BOOL ;
   _X_TEL_POS_4 : BOOL ;
   _X_TEL_POS_5 : BOOL ;
   _X_TEL_POS_6 : BOOL ;
   _X_TEL_POS_7 : BOOL ;
   _X_TEL_POS_8 : BOOL ;
   _X_TEL_POS_9 : BOOL ;
   _X_TEL_POS_10 : BOOL ;
   _X_TEL_POS_11 : BOOL ;
   _X_TEL_POS_12 : BOOL ;
  END_STRUCT ;	
BEGIN
   _di.MotorTargPos := L#10000;
   _di.MotorActPos := L#10000;
   _di.SwsMin := L#9125;
   _di.SwsMax := L#10860;
   _di.PresetPos := L#10000;
   _di.AreaWin := L#80;
   _di.PosWin := L#1;
   _di.SlowWin := L#50;
   _di.StopWin := L#1;
   _di.ValPosCenter := L#10000;
   _di.ValActPos1 := L#10424;
   _di.ValActPos2 := L#10774;
   _di.VolPosInternHook := L#10505;
   _di.ValueLastCycle := L#10000;
   _di.ManPrevPos := L#9535;
   _di.ManActPos := L#10000;
   _di.ManNextPos := L#10000;
   _di.ManMinPos := L#9155;
   _di.ManMaxPos := L#10000;
   _di.ManTargPos := L#10000;
   _di._26 := L#10407;
   _di._27 := L#10729;
   _di._Enco_Helpflag1 := L#10;
   _di._Enco_Helpflag2 := L#-10;
   _di._ActEncoder_mm := L#2000;
   _di._PresetEncoder_mm := L#2000;
   _di._FactorEncoder := L#73;
   _di._Enc_Korrektur := L#2000;
   _di._Enc_Window := L#10;
   _di.ActPosMinusOffset := L#10000;
   _di._Pos_Center := L#2000;
   _di._Pos_left_big := L#3090;
   _di._Pos_left_mid := L#2950;
   _di._Pos_left_small_1 := L#2670;
   _di._Pos_left_small_2 := L#3030;
   _di._Pos_right_big := L#900;
   _di._Pos_right_mid := L#1040;
   _di._Pos_right_small_1 := L#1320;
   _di._Pos_right_small_2 := L#960;
   _i.TargPosNo := 1;
   _i.ActAreaNo := 620;
   _i.ActPosNo := 620;
   _i.ActValueMeasureDiameter := 549;
   _i._40 := 15;
   _i._41 := 1789;
   _i._42 := 739;
   _i._43 := 482;
   _i._44 := 1910;
   _i._46 := 3455;
   _i._47 := 1787;
   _i._48 := 733;
   _i._49 := 480;
   _i._50 := 1908;
   _i._51 := 2808;
   _x.RelForPos := TRUE;
   _x.InArea := TRUE;
   _x.InPosCenter := TRUE;
   _x.InAreaCenter := TRUE;
   _x.ScanInPos := TRUE;
   _x.Free := TRUE;
   _x.AutoPosOk := TRUE;
   _x.BuffOccOK := TRUE;
   _x.ReleasePlus := TRUE;
   _x.ReleaseMinus := TRUE;
   _x.PosCenterChk := TRUE;
   _x.BuffFree := TRUE;
   _x.Free_Steute := TRUE;
   _x._95 := TRUE;
   _x.InPosition := TRUE;
END_DATA_BLOCK

DATA_BLOCK "DB_BRI"	// DB 5
VERSION : 0.1
  STRUCT
   _di : STRUCT
    MotorTargPos : DINT ;
    MotorActPos : DINT ;
    SwsMin : DINT ;
    SwsMax : DINT ;
    PresetPos : DINT ;
    PresetData : DINT ;
    AreaWin : DINT ;
    PosWin : DINT ;
    _08 : DINT ;
    _09 : DINT ;
    _10 : DINT ;
    _11 : DINT ;
    _12 : DINT ;
    _13 : DINT ;
    _14 : DINT ;
    _15 : DINT ;
    _16 : DINT ;
    _17 : DINT ;
    _18 : DINT ;
    Offset : DINT ;
    ManPrevPos : DINT ;
    ManActPos : DINT ;
    ManNextPos : DINT ;
    ManMinPos : DINT ;
    ManMaxPos : DINT ;
    ManTargPosVal : DINT ;
    _26 : DINT ;
    _27 : DINT ;
    _28 : DINT ;
    _29 : DINT ;
    _30 : DINT ;
    _31 : DINT ;
    _32 : DINT ;
    _33 : DINT ;
    _34 : DINT ;
    ActPosMinusOffset : DINT ;
    TargPosPlusOffset : DINT ;
    _37 : DINT ;
    _38 : DINT ;
    _39 : DINT ;
    _40 : DINT ;
    _41 : DINT ;
    _42 : DINT ;
    _43 : DINT ;
    _44 : DINT ;
    _45 : DINT ;
    _46 : DINT ;
    _47 : DINT ;
    _48 : DINT ;
    _49 : DINT ;
    _50 : DINT ;
    _51 : DINT ;
    _52 : DINT ;
    _53 : DINT ;
    _54 : DINT ;
    _55 : DINT ;
    _56 : DINT ;
    _57 : DINT ;
    _58 : DINT ;
    _59 : DINT ;
    _60 : DINT ;
    _61 : DINT ;
    _62 : DINT ;
    _63 : DINT ;
    _64 : DINT ;
    _65 : DINT ;
    _66 : DINT ;
    _67 : DINT ;
    _68 : DINT ;
    _69 : DINT ;
    _70 : DINT ;
    _71 : DINT ;
    _72 : DINT ;
    _73 : DINT ;
    _74 : DINT ;
   END_STRUCT ;
   _i : STRUCT
    MotorIn_00 : INT ;
    MotorIn_01 : INT ;
    MotorIn_02 : INT ;
    MotorIn_03 : INT ;
    MotorIn_04 : INT ;
    MotorIn_05 : INT ;
    MotorOut_00 : INT ;
    MotorOut_01 : INT ;
    MotorOut_02 : INT ;
    MotorOut_03 : INT ;
    MotorOut_04 : INT ;
    MotorOut_05 : INT ;
    MotorCrtWord : INT ;
    MotorTargSpeed : INT ;
    MotorTargAcc : INT ;
    MotorTargDeacc : INT ;
    MotorStateWord : INT ;
    MotorActSpeed : INT ;
    MotorActCurrent : INT ;
    MotorActWorkLoad : INT ;
    SourcePosNo : INT ;
    TargPosNo : INT ;
    ActAreaNo : INT ;
    ServiceV : INT ;
    ManualV : INT ;
    OnlineV : INT ;
    ForcedSlowV : INT ;
    RuntimeSec : INT ;
    ActPosNo : INT ;
    ScanAreaNo : INT ;
    SpeedManual : INT ;
    SafetySpeed : INT ;	//sichere Geschwindigkeit (1/min)
    SpeedForcSlow : INT ;
    SpeedManSlo : INT ;
    Acceleration : INT ;
    Deacceleration : INT ;
    _36 : INT ;
    ManTargPosNo : INT ;
    PrevPosNo : INT ;
    NextPosNo : INT ;
    MinPosNo : INT ;
    MaxPosNo : INT ;
    _42 : INT ;
    _43 : INT ;
    _44 : INT ;
    ActLIF_DBNo : INT ;
    _46 : INT ;
    _47 : INT ;
    _48 : INT ;
    _49 : INT ;
    _50 : INT ;
    _51 : INT ;
    _52 : INT ;
    _53 : INT ;
    _54 : INT ;
    _55 : INT ;
    _56 : INT ;
    _57 : INT ;
    _58 : INT ;
    _59 : INT ;
    _60 : INT ;
    _61 : INT ;
    _62 : INT ;
    _63 : INT ;
    _64 : INT ;
    _65 : INT ;
    _66 : INT ;
    _67 : INT ;
    _68 : INT ;
    _69 : INT ;
    _70 : INT ;
    _71 : INT ;
    _72 : INT ;
    _73 : INT ;
    _74 : INT ;
    _75 : INT ;
    _76 : INT ;
    _77 : INT ;
    _78 : INT ;
    _79 : INT ;
    _80 : INT ;
    _81 : INT ;
    _82 : INT ;
    _83 : INT ;
    _84 : INT ;
    _85 : INT ;
    _86 : INT ;
    _87 : INT ;
    _88 : INT ;
    _89 : INT ;
    _90 : INT ;
    _91 : INT ;
    _92 : INT ;
    _93 : INT ;
    _94 : INT ;
    _95 : INT ;
    _96 : INT ;
    _97 : INT ;
    _98 : INT ;
    DriveErrorCode : INT ;
   END_STRUCT ;
   _x : STRUCT
    InchMinus : BOOL ;
    InchPlus : BOOL ;
    TargIsPos : BOOL ;
    RelForPos : BOOL ;
    MovesMinus : BOOL ;
    MovesPlus : BOOL ;
    Moves : BOOL ;
    InArea : BOOL ;
    InPos : BOOL ;
    FastStop : BOOL ;
    ManPosFound : BOOL ;
    MotorReady : BOOL ;
    MotorRefOk : BOOL ;
    ForcedSlow : BOOL ;
    StartPos : BOOL ;
    Position_Found : BOOL ;
    pFl_StartPos : BOOL ;
    _17 : BOOL ;
    DelayFaststop : BOOL ;
    ReleaseScan : BOOL ;
    ScanInPos : BOOL ;
    AutoInPos : BOOL ;
    TargPosFront : BOOL ;
    TargPosBack : BOOL ;
    InPosCart : BOOL ;
    _25 : BOOL ;
    _26 : BOOL ;
    _27 : BOOL ;
    _28 : BOOL ;
    _29 : BOOL ;
    _30 : BOOL ;
    _31 : BOOL ;
    _32 : BOOL ;
    _33 : BOOL ;
    _34 : BOOL ;
    _35 : BOOL ;
    _36 : BOOL ;
    _37 : BOOL ;
    _38 : BOOL ;
    _39 : BOOL ;
    _40 : BOOL ;
    _41 : BOOL ;
    _42 : BOOL ;
    _43 : BOOL ;
    _44 : BOOL ;
    _45 : BOOL ;
    _46 : BOOL ;
    _47 : BOOL ;
    _48 : BOOL ;
    _49 : BOOL ;
    _50 : BOOL ;
    PresetOffset : BOOL ;
    _52 : BOOL ;
    _53 : BOOL ;
    _54 : BOOL ;
    _55 : BOOL ;
    _56 : BOOL ;
    _57 : BOOL ;
    _58 : BOOL ;
    _59 : BOOL ;
    _60 : BOOL ;
    _61 : BOOL ;
    fs_Minus_SW : BOOL ;	//forced slow software
    fs_Plus_Sw : BOOL ;	//forced slow software
    _64 : BOOL ;
    _65 : BOOL ;
    _66 : BOOL ;
    _67 : BOOL ;
    _68 : BOOL ;
    _69 : BOOL ;
    _70 : BOOL ;
    _71 : BOOL ;
    _72 : BOOL ;
    _73 : BOOL ;
    _74 : BOOL ;
    _75 : BOOL ;
    _76 : BOOL ;
    _77 : BOOL ;
    _78 : BOOL ;
    _79 : BOOL ;
    _80 : BOOL ;
    _81 : BOOL ;
    _82 : BOOL ;
    _83 : BOOL ;
    _84 : BOOL ;
    _85 : BOOL ;
    _86 : BOOL ;
    _87 : BOOL ;
    _88 : BOOL ;
    _89 : BOOL ;
    _90 : BOOL ;
    _91 : BOOL ;
    _92 : BOOL ;
    _93 : BOOL ;
    _94 : BOOL ;
    _95 : BOOL ;
   END_STRUCT ;
  END_STRUCT ;	
BEGIN
   _di.MotorTargPos := L#2000;
   _di.MotorActPos := L#2000;
   _di.SwsMin := L#330;
   _di.SwsMax := L#7000;
   _di.AreaWin := L#10;
   _di.PosWin := L#1;
   _di._08 := L#2000;
   _di.ManPrevPos := L#5134;
   _di.ManActPos := L#7046;
   _di.ManNextPos := L#9344;
   _di.ManMinPos := L#1313;
   _di.ManMaxPos := L#9344;
   _di.ManTargPosVal := L#3223;
   _di.ActPosMinusOffset := L#2000;
   _di.TargPosPlusOffset := L#2000;
   _i.MotorIn_00 := 526;
   _i.MotorIn_02 := 2000;
   _i.MotorOut_00 := 6144;
   _i.MotorOut_02 := 2000;
   _i.MotorOut_03 := 1160;
   _i.MotorOut_04 := 2600;
   _i.MotorOut_05 := 2600;
   _i.MotorCrtWord := 6144;
   _i.MotorTargSpeed := 1160;
   _i.MotorTargAcc := 2600;
   _i.MotorTargDeacc := 2600;
   _i.MotorStateWord := 526;
   _i.TargPosNo := 6;
   _i.ActAreaNo := 4;
   _i.ServiceV := 1;
   _i.ManualV := 30;
   _i.OnlineV := 100;
   _i.ForcedSlowV := 5;
   _i.ActPosNo := 6;
   _i.ScanAreaNo := 5;
   _i.SpeedManual := 2;
   _i.SpeedForcSlow := 5;
   _i.SpeedManSlo := 2;
   _i.Acceleration := 3000;
   _i.Deacceleration := 3000;
   _i._36 := 2;
   _i.ManTargPosNo := 2;
   _i.PrevPosNo := 3;
   _i.NextPosNo := 5;
   _i.MinPosNo := 1;
   _i.MaxPosNo := 5;
   _i.ActLIF_DBNo := 201;
   _i.DriveErrorCode := 2;
   _x.InArea := TRUE;
   _x.FastStop := TRUE;
   _x.MotorReady := TRUE;
   _x.MotorRefOk := TRUE;
   _x.Position_Found := TRUE;
   _x.ScanInPos := TRUE;
   _x.AutoInPos := TRUE;
END_DATA_BLOCK

DATA_BLOCK "DB_ComGateway"	// DB 10
VERSION : 0.1
  STRUCT
   TM : STRUCT
    StateWord : INT ;
    TotalLength : INT ;
    FaceLength : INT ;
    Circum : INT ;
    BriActPos : INT ;
    TroActPos : INT ;
    LifActPos : INT ;
    TelActPos : INT ;
    WidActPos : INT ;
    Ax05ActPos : INT ;
    Ax06ActPos : INT ;
    Ax07ActPos : INT ;
    Ax08ActPos : INT ;
    Ax09ActPos : INT ;
    BriMotorPos : DINT ;
    TroMotorPos : DINT ;
    LifMotorPos : DINT ;
    TelMotorPos : DINT ;
    WidMotorPos : DINT ;
    Ax05MotorPos : DINT ;
    Ax06MotorPos : DINT ;
    Ax07MotorPos : DINT ;
    Ax08MotorPos : DINT ;
    Ax09MotorPos : DINT ;
    ParaCnt : INT ;
    ParaNo : INT ;
    ParaData : DINT ;
    Err00 : INT ;
    Err01 : INT ;
    Err02 : INT ;
    Err03 : INT ;
    Err04 : INT ;
    Err05 : INT ;
    Err06 : INT ;
    Err07 : INT ;
    Err08 : INT ;
    Err09 : INT ;
    Err10 : INT ;
    Err11 : INT ;
    StepNo : INT ;
    WorkHours : DINT ;
    _53 : INT ;
    _54 : INT ;
    CommCounterToMaster : INT ;
    _56 : INT ;
    _57 : INT ;
    _58 : INT ;
    InvStateWord : INT ;
    Lifebit : BOOL ;
    TeleskopsFree : BOOL ;
    Buffer_Free : BOOL ;
    LiftTop : BOOL ;
    Online : BOOL ;
    ReadyOnline : BOOL ;
    Error : BOOL ;
    MovingSource : BOOL ;
    MovingTarget : BOOL ;
    TeleskopCenterpos : BOOL ;
    OrderRunning : BOOL ;
    OrderEnd : BOOL ;
    OrderPaused : BOOL ;
    Bit13 : BOOL ;
    TargetNok : BOOL ;
    RequestTurne : BOOL ;
    Spare122 : WORD ;
    Spare124 : WORD ;
    Spare126 : WORD ;
    Move : UDT 7;
    Spare154 : WORD ;
    Spare156 : WORD ;
    Spare158 : WORD ;
    ErrorCabinet : STRUCT
     Err00 : INT ;
     Err01 : INT ;
     Err02 : INT ;
     Err03 : INT ;
     Err04 : INT ;
     Err05 : INT ;
     Err06 : INT ;
     Err07 : INT ;
     Err08 : INT ;
     Err09 : INT ;
     Err10 : INT ;
     Err11 : INT ;
    END_STRUCT ;
    LS_1 : STRUCT
     SPARE_00 : BOOL ;
     SPARE_01 : BOOL ;
     SPARE_02 : BOOL ;
     SPARE_03 : BOOL ;
     SPARE_04 : BOOL ;
     SPARE_05 : BOOL ;
     Online : BOOL ;
     Ready : BOOL ;
     Palette_In_Station : BOOL ;
     Pos_11_Free : BOOL ;
     Pos_12_Free : BOOL ;
     SPARE_13 : BOOL ;
     SPARE_14 : BOOL ;
     SPARE_15 : BOOL ;
     SPARE_16 : BOOL ;
     SPARE_17 : BOOL ;
    END_STRUCT ;
    LS_2 : STRUCT
     SPARE_00 : BOOL ;
     SPARE_01 : BOOL ;
     SPARE_02 : BOOL ;
     SPARE_03 : BOOL ;
     SPARE_04 : BOOL ;
     SPARE_05 : BOOL ;
     Online : BOOL ;
     Ready : BOOL ;
     Palette_In_Station : BOOL ;
     Pos_11_Free : BOOL ;
     Pos_12_Free : BOOL ;
     SPARE_13 : BOOL ;
     SPARE_14 : BOOL ;
     SPARE_15 : BOOL ;
     SPARE_16 : BOOL ;
     SPARE_17 : BOOL ;
    END_STRUCT ;
    LS_3 : STRUCT
     SPARE_00 : BOOL ;
     SPARE_01 : BOOL ;
     SPARE_02 : BOOL ;
     SPARE_03 : BOOL ;
     SPARE_04 : BOOL ;
     SPARE_05 : BOOL ;
     Online : BOOL ;
     Ready : BOOL ;
     Palette_In_Station : BOOL ;
     Pos_11_Free : BOOL ;
     Pos_12_Free : BOOL ;
     SPARE_13 : BOOL ;
     SPARE_14 : BOOL ;
     SPARE_15 : BOOL ;
     SPARE_16 : BOOL ;
     SPARE_17 : BOOL ;
    END_STRUCT ;
    Spare : ARRAY  [1 .. 5 ] OF WORD ;
   END_STRUCT ;
   FM : STRUCT
    ReleaseManual : BOOL ;
    spare01 : BOOL ;
    StartOrder : BOOL ;
    CleareOrder : BOOL ;
    StopOrder : BOOL ;
    spare05 : BOOL ;
    spare06 : BOOL ;
    ReleaseOnline : BOOL ;
    Lifebit : BOOL ;
    spare11 : BOOL ;
    StartBasePos : BOOL ;
    ChangeOrder : BOOL ;
    QuitOrderFinished : BOOL ;
    ResetErrors : BOOL ;
    ServiceOn : BOOL ;
    BypassLimmitsOn : BOOL ;
    TotalLength : INT ;
    FaceLength : INT ;
    Circum : INT ;
    SourceBri : INT ;
    SourceTro : INT ;
    SourceLif : INT ;
    SourceTel : INT ;
    SourceAx04 : INT ;
    SourceAx05 : INT ;
    SourceAx06 : INT ;
    SourceAx07 : INT ;
    SourceAx08 : INT ;
    SourceAx09 : INT ;
    TargBri : INT ;
    TargTro : INT ;
    TargLif : INT ;
    TargTel : INT ;
    TargAx04 : INT ;
    TargAx05 : INT ;
    TargAx06 : INT ;
    TargAx07 : INT ;
    TargAx08 : INT ;
    TargAx09 : INT ;
    Occ00 : INT ;
    Occ01 : INT ;
    Occ02 : INT ;
    Occ03 : INT ;
    SafetyAreas00 : INT ;
    SafetyAreas01 : INT ;
    ParaCnt : INT ;
    ParaNo : INT ;
    ParaData : DINT ;
    _34 : INT ;
    _35 : INT ;
    _36 : INT ;
    _37 : INT ;
    _38 : INT ;
    _39 : INT ;
    _40 : INT ;
    _41 : INT ;
    _42 : INT ;
    _43 : INT ;
    _44 : INT ;
    CommCounterFromMaster : INT ;
    _46 : INT ;
    _47 : INT ;
    _48 : INT ;
    InvCrtWord : INT ;
    Bit100_0 : BOOL ;
    Bit100_1 : BOOL ;
    Bit100_2 : BOOL ;
    Bit100_3 : BOOL ;
    Bit100_4 : BOOL ;
    Bit100_5 : BOOL ;
    Bit00_6 : BOOL ;
    Bit100_7 : BOOL ;
    Release : BOOL ;
    BypassLimits : BOOL ;
    Service : BOOL ;
    Sw_Manual : BOOL ;
    Bit101_4 : BOOL ;
    Bit101_5 : BOOL ;
    Bit101_6 : BOOL ;
    Bit101_7 : BOOL ;
    BrPosRelease : INT ;
    TrPosRelease : INT ;
    LiPosRelease : INT ;
    TlPosRelease : INT ;
    spare_110 : INT ;
    spare_112 : INT ;
    spare_114 : INT ;
    spare_116 : INT ;
    spare_118 : INT ;
    spare_120 : INT ;
    spare_122 : INT ;
    spare_124 : INT ;
    spare_126 : INT ;
    Move : UDT 7;
    LS_1 : STRUCT
     Start_Load : BOOL ;
     Start_Unload : BOOL ;
     Step_Load : BOOL ;
     Step_Unload : BOOL ;
     CleareOrder : BOOL ;
     SPARE_05 : BOOL ;
     SPARE_06 : BOOL ;
     SPARE_07 : BOOL ;
     SPARE_10 : BOOL ;
     SPARE_11 : BOOL ;
     SPARE_12 : BOOL ;
     SPARE_13 : BOOL ;
     SPARE_14 : BOOL ;
     SPARE_15 : BOOL ;
     SPARE_16 : BOOL ;
     SPARE_17 : BOOL ;
     TotalLength : INT ;
     FaceLength : INT ;
     Circum : INT ;
    END_STRUCT ;
    Spare : ARRAY  [1 .. 19 ] OF WORD ;
   END_STRUCT ;
  END_STRUCT ;	
BEGIN
   TM.StateWord := 1170;
   TM.BriActPos := 5;
   TM.TroActPos := 8;
   TM.LifActPos := 2;
   TM.TelActPos := 100;
   TM.BriMotorPos := L#24802;
   TM.TroMotorPos := L#25010;
   TM.LifMotorPos := L#5859;
   TM.TelMotorPos := L#2000;
   TM.StepNo := 1050;
   TM.CommCounterToMaster := 4163;
   TM.TeleskopsFree := TRUE;
   TM.Online := TRUE;
   TM.MovingSource := TRUE;
   TM.OrderRunning := TRUE;
   TM.Move.Action := 4;
   TM.Move.Value_01 := 5;
   TM.Move.Value_02 := 8;
   TM.Move.Value_03 := 100;
   TM.Move.Value_04 := 100;
   TM.LS_1.Online := TRUE;
   TM.LS_1.Ready := TRUE;
   TM.LS_1.Palette_In_Station := TRUE;
   TM.LS_1.Pos_11_Free := TRUE;
   TM.LS_1.Pos_12_Free := TRUE;
   TM.LS_2.Online := TRUE;
   TM.LS_2.Ready := TRUE;
   TM.LS_2.Palette_In_Station := TRUE;
   TM.LS_2.Pos_11_Free := TRUE;
   TM.LS_2.Pos_12_Free := TRUE;
   TM.LS_3.Online := TRUE;
   TM.LS_3.Ready := TRUE;
   TM.LS_3.Palette_In_Station := TRUE;
   TM.LS_3.Pos_11_Free := TRUE;
   TM.LS_3.Pos_12_Free := TRUE;
   TM.Spare[1] := W#16#4241;
   TM.Spare[2] := W#16#5545;
   TM.Spare[3] := W#16#5520;
   FM.TotalLength := 2300;
   FM.Circum := 630;
   FM.SourceBri := 5;
   FM.SourceTro := 8;
   FM.SourceLif := 2;
   FM.SourceTel := 1;
   FM.TargAx04 := 11301;
   FM.ParaCnt := 321;
   FM.ParaNo := 654;
   FM.ParaData := L#76542;
   FM.CommCounterFromMaster := 4162;
   FM.Bit100_1 := TRUE;
   FM.Bit100_2 := TRUE;
   FM.Move.MsgCounter := 648;
   FM.Move.Action := 4;
   FM.Move.Value_01 := 5;
   FM.Move.Value_02 := 8;
   FM.Move.Value_03 := 100;
   FM.Move.Value_04 := 100;
END_DATA_BLOCK

DATA_BLOCK "IDB_FB2_TRO"	// DB 12
AUTHOR : Koenig
VERSION : 0.0
"MovidriveB_Control"
BEGIN
END_DATA_BLOCK

DATA_BLOCK "IDB_FB2_LIF"	// DB 13
AUTHOR : Koenig
VERSION : 0.0
"MovidriveB_Control"
BEGIN
END_DATA_BLOCK

DATA_BLOCK "IDB_FB21_TEL"	// DB 14
VERSION : 0.0
"CheckEncoder"
BEGIN
END_DATA_BLOCK

DATA_BLOCK "DB_OrderBuffer"	// DB 15
VERSION : 0.1
  STRUCT
   SourceBri : INT ;
   SourceTro : INT ;
   SourceLif : INT ;
   SourceTel : INT ;
   TargetBri : INT ;
   TargetTro : INT ;
   TargetLif : INT ;
   TargetTel : INT ;
   OrderTotalLength : INT ;
   OrderFaceLength : INT ;
   OrderCircum : INT ;
  END_STRUCT ;	
BEGIN
   SourceBri := 5;
   SourceTro := 8;
   SourceLif := 2;
   SourceTel := 1;
   OrderTotalLength := 2300;
   OrderCircum := 630;
END_DATA_BLOCK

DATA_BLOCK "DB_IntentData"	// DB 17
VERSION : 0.1
  STRUCT
   BRI : STRUCT
    PosNo : INT ;
    PosVal : DINT ;
   END_STRUCT ;
   TRO : STRUCT
    PosNo : INT ;
    PosVal : DINT ;
   END_STRUCT ;
   LIF : STRUCT
    PosNo : INT ;
    PosVal : DINT ;
   END_STRUCT ;
   TEL : STRUCT
    PosNo : INT ;
    PosVal : DINT ;
   END_STRUCT ;
   Axis5 : STRUCT
    PosNo : INT ;
    PosVal : DINT ;
   END_STRUCT ;
   Axis6 : STRUCT
    PosNo : INT ;
    PosVal : DINT ;
   END_STRUCT ;
   Axis7 : STRUCT
    PosNo : INT ;
    PosVal : DINT ;
   END_STRUCT ;
   Axis8 : STRUCT
    PosNo : INT ;
    PosVal : DINT ;
   END_STRUCT ;
   Axis9 : STRUCT
    PosNo : INT ;
    PosVal : DINT ;
   END_STRUCT ;
   Axis10 : STRUCT
    PosNo : INT ;
    PosVal : DINT ;
   END_STRUCT ;
   Hookdata : UDT 102;
   LIF_DB_1 : INT ;
   LIF_DB_2 : INT ;
  END_STRUCT ;	
BEGIN
   BRI.PosNo := 2;
   BRI.PosVal := L#18161;
   TRO.PosNo := 1;
   LIF.PosNo := 1;
   TEL.PosNo := 100;
   Hookdata.HookOver := L#10020;
   Hookdata.TelPos_1.HookType := 1;
   Hookdata.TelPos_1.TotLengthMin := 1100;
   Hookdata.TelPos_1.TotLengthMax := 1100;
   Hookdata.TelPos_1.FaceLengthMax := 1100;
   Hookdata.TelPos_1.CircumMax := 662;
   Hookdata.TelPos_1.TelPos := L#8419;
   Hookdata.TelPos_1.Reserve1 := 3;
   LIF_DB_1 := 321;
   LIF_DB_2 := 331;
END_DATA_BLOCK

DATA_BLOCK "DB_TargetData"	// DB 19
VERSION : 0.1
  STRUCT
   BrPosNo : INT  := 1;
   BrPosVal : DINT  := L#1000;
   TrPosNo : INT  := 1;
   TrPosVal : DINT ;
   LiPosNo : INT ;
   LiPosValHo : DINT ;
   LiPosValHu : DINT ;
   TlPosNo : INT ;
   TlPosVal : DINT ;
   Hooktype : INT ;
   CircumMax : INT ;
   Reserve : INT ;
   Hookdata : UDT 102;
  END_STRUCT ;	
BEGIN
   BrPosNo := 5;
   BrPosVal := L#4160;
   TrPosNo := 8;
   TrPosVal := L#160212;
   LiPosNo := 2;
   LiPosValHo := L#5745;
   LiPosValHu := L#5860;
   TlPosNo := 1;
   TlPosVal := L#3;
   Hookdata.HookOver := L#5745;
   Hookdata.HookUnderOffset := L#115;
   Hookdata.TelPos_1.TelPos := L#3;
END_DATA_BLOCK

DATA_BLOCK "IDB_FB22"	// DB 22
VERSION : 0.0
"GetCircumference"
BEGIN
END_DATA_BLOCK

DATA_BLOCK "IDB_FB29"	// DB 29
VERSION : 0.0
"WAGO_Analog_Input_4_20"
BEGIN
END_DATA_BLOCK

DATA_BLOCK "IDB_MasterInterface"	// DB 33
VERSION : 0.0
"MasterInterface"
BEGIN
END_DATA_BLOCK

DATA_BLOCK "DB_ANALOG"	// DB 50
VERSION : 0.1
  STRUCT
   Adress : INT  := 272;
   OutputMax : INT  := 4095;	//maximaler Integerwert AD-Wandler füe Meßbereich
   RangeBegin : INT  := 400;	//Meßbereich Anfang Sensor (mm)
   RangeEnd : INT ;	//Meßbereich Anfang Ende (mm)
   DiamCyl : INT ;	//Zylinderdurchmesser
   CircumCyl : INT ;	//Zylinderumfang
   ReferenzValue : INT  := 431;	//Referenzwert
   CircumRef : INT  := 50;	//Umfang Referenzzylinder
   Statusbit_0 : BOOL ;	//Messbereichunterschreitung
   Statusbit_1 : BOOL ;	//Messbereichsüberschreitung/Leitungsbruch
   Statusbit_2 : BOOL ;	//Messbereichsüberschreitung/Leitungsbruch
   enable : BOOL ;
   preset : BOOL ;
   bit_14_5 : BOOL ;
   bit_14_6 : BOOL ;
   bit_14_7 : BOOL ;
  END_STRUCT ;	
BEGIN
   Adress := 272;
   OutputMax := 4095;
   RangeBegin := 100;
   RangeEnd := 500;
   DiamCyl := -137;
   CircumCyl := -431;
   ReferenzValue := 431;
   CircumRef := 50;
   enable := TRUE;
END_DATA_BLOCK

